CASE THIS^.stSeqCtrlGeneral.eActiveSeqState OF
E_SEQ_GENERAL.READY:;

	
E_SEQ_GENERAL.EXECUTE:;
	IF TRUE
	THEN
		THIS^.stSeqCtrlGeneral.eActiveSeqState := E_SEQ_GENERAL.RESET;
	END_IF
  
E_SEQ_GENERAL.RESET:;
	stSeqCtrlGeneral.iInternalSeqStateCase := 0;
	IF TRUE
	THEN
		THIS^.stSeqCtrlGeneral.eActiveSeqState := E_SEQ_GENERAL.BUSY;
	END_IF
  
E_SEQ_GENERAL.BUSY:;
	CASE THIS^.stSeqCtrlGeneral.iInternalSeqStateCase OF
    0:  // Check state
      IF TRUE
      AND THIS^.itfSensorOpened.P_Active 
      AND THIS^.itfSensorClosed.P_Active 
			THEN 
        THIS^.stSeqCtrlGeneral.eActiveSeqState := E_SEQ_GENERAL.ERROR;
      ELSIF TRUE
      AND THIS^.itfSensorClosed.P_Active
      THEN
        THIS^.stSeqCtrlGeneral.iInternalSeqStateCase := 1000;
      ELSE
        THIS^.itfClose.M_Set();
        THIS^.itfOpen.M_Reset();
        THIS^.stSeqCtrlGeneral.iInternalSeqStateCase := 10;
			END_IF
      
    10: // wait for the end position sensor
      IF TRUE 
			THEN 
        IF TRUE
        AND THIS^.itfSensorClosed.P_Active
        THEN
          THIS^.itfClose.M_Reset();
          THIS^.stSeqCtrlGeneral.iInternalSeqStateCase := 1000;
				END_IF
			END_IF
      
	ELSE
		THIS^.stSeqCtrlGeneral.eActiveSeqState := E_SEQ_GENERAL.DONE;  
	END_CASE
	THIS^.stSeqCtrlGeneral.strExtraInfo := CONCAT('Internal state: ', TO_STRING(THIS^.stSeqCtrlGeneral.iInternalSeqStateCase));

E_SEQ_GENERAL.DONE:;

E_SEQ_GENERAL.ERROR:;

E_SEQ_GENERAL.TIME_OUT:; 
IF TRUE
AND THIS^.stSeqCtrlGeneral.bTimeOutActiveQuit 
THEN
  THIS^.stSeqCtrlGeneral.strExtraInfo := 'Bitte quittieren und erneut testen';
  IF TRUE
  //AND itfOpMode.P_QUIT
  THEN
    THIS^.stSeqCtrlGeneral.eActiveSeqState := E_SEQ_GENERAL.EXECUTE;
	END_IF
  
END_IF

ELSE
  THIS^.stSeqCtrlGeneral.eActiveSeqState := E_SEQ_GENERAL.ERROR;
END_CASE
END_METHOD

METHOD PRIVATE _m_Seq_INIT : BOOL
VAR
  ActiveSeq: STRING;
END_VAR
//THIS^._m_GeneralStepSetting(StepType:=E_STEP_STATE_TYPE.INIT,
ActiveSeq := TO_STRING(THIS^.eSeq);

CASE THIS^.stSeqCtrlGeneral.eActiveSeqState OF
E_SEQ_GENERAL.READY:;

	
E_SEQ_GENERAL.EXECUTE:;
	IF TRUE
	THEN
		THIS^.stSeqCtrlGeneral.eActiveSeqState := E_SEQ_GENERAL.RESET;
	END_IF
  
E_SEQ_GENERAL.RESET:;
	stSeqCtrlGeneral.iInternalSeqStateCase := 0;
	IF TRUE
	THEN
		THIS^.stSeqCtrlGeneral.eActiveSeqState := E_SEQ_GENERAL.BUSY;
	END_IF
  
E_SEQ_GENERAL.BUSY:;
	CASE THIS^.stSeqCtrlGeneral.iInternalSeqStateCase OF
    0:  // Reset valve
      IF TRUE 
			THEN 
        IF THIS^.bNC THEN
          THIS^.itfClose.M_Set();
          THIS^.itfOpen.M_Reset();
        ELSE
          THIS^.itfClose.M_Reset();
          THIS^.itfOpen.M_Set();
				END_IF
        THIS^.stSeqCtrlGeneral.iInternalSeqStateCase := 10;
			END_IF
      
    10: // Wait for the end position sensor
      IF TRUE 
			THEN 
        IF THIS^.bNC 
        AND THIS^.itfSensorClosed.P_Active 
        THEN
          THIS^.itfClose.M_Reset();
          THIS^.stSeqCtrlGeneral.iInternalSeqStateCase := 1000;
        ELSIF NOT THIS^.bNC
        AND THIS^.itfSensorOpened.P_Active
        THEN
          THIS^.itfOpen.M_Reset();
          THIS^.stSeqCtrlGeneral.iInternalSeqStateCase := 1000;
				END_IF
			END_IF
      
	ELSE
		THIS^.stSeqCtrlGeneral.eActiveSeqState := E_SEQ_GENERAL.DONE;  
	END_CASE
	THIS^.stSeqCtrlGeneral.strExtraInfo := CONCAT('Internal state: ', TO_STRING(THIS^.stSeqCtrlGeneral.iInternalSeqStateCase));

E_SEQ_GENERAL.DONE:;

E_SEQ_GENERAL.ERROR:;

E_SEQ_GENERAL.TIME_OUT:; 
IF TRUE
AND THIS^.stSeqCtrlGeneral.bTimeOutActiveQuit 
THEN
  THIS^.stSeqCtrlGeneral.strExtraInfo := 'Bitte quittieren und erneut testen';
  IF TRUE
  //AND itfOpMode.P_QUIT
  THEN
    THIS^.stSeqCtrlGeneral.eActiveSeqState := E_SEQ_GENERAL.EXECUTE;
	END_IF
  
END_IF

ELSE
  THIS^.stSeqCtrlGeneral.eActiveSeqState := E_SEQ_GENERAL.ERROR;
END_CASE
END_METHOD

METHOD PRIVATE _m_Seq_OPEN : BOOL
VAR
  ActiveSeq: STRING;
END_VAR
//THIS^._m_GeneralStepSetting(StepType:=E_STEP_STATE_TYPE.INIT,
ActiveSeq := TO_STRING(THIS^.eSeq);

CASE THIS^.stSeqCtrlGeneral.eActiveSeqState OF
E_SEQ_GENERAL.READY:;

	
E_SEQ_GENERAL.EXECUTE:;
	IF TRUE
	THEN
		THIS^.stSeqCtrlGeneral.eActiveSeqState := E_SEQ_GENERAL.RESET;
	END_IF
  
E_SEQ_GENERAL.RESET:;
	stSeqCtrlGeneral.iInternalSeqStateCase := 0;
	IF TRUE
	THEN
		THIS^.stSeqCtrlGeneral.eActiveSeqState := E_SEQ_GENERAL.BUSY;
	END_IF
  
E_SEQ_GENERAL.BUSY:;
	CASE THIS^.stSeqCtrlGeneral.iInternalSeqStateCase OF
    0:  // Check state
      IF TRUE
      AND THIS^.itfSensorOpened.P_Active 
      AND THIS^.itfSensorClosed.P_Active 
			THEN 
        THIS^.stSeqCtrlGeneral.eActiveSeqState := E_SEQ_GENERAL.ERROR;
      ELSIF TRUE
      AND THIS^.itfSensorOpened.P_Active
      THEN
        THIS^.stSeqCtrlGeneral.iInternalSeqStateCase := 1000;
      ELSE
        THIS^.itfClose.M_Reset();
        THIS^.itfOpen.M_Set();
        THIS^.stSeqCtrlGeneral.iInternalSeqStateCase := 10;
			END_IF
      
    10: // wait for the end position sensor
      IF TRUE 
			THEN 
        IF TRUE
        AND THIS^.itfSensorOpened.P_Active
        THEN
          THIS^.itfOpen.M_Reset();
          THIS^.stSeqCtrlGeneral.iInternalSeqStateCase := 1000;
				END_IF
			END_IF
      
	ELSE
		THIS^.stSeqCtrlGeneral.eActiveSeqState := E_SEQ_GENERAL.DONE;  
	END_CASE
	THIS^.stSeqCtrlGeneral.strExtraInfo := CONCAT('Internal state: ', TO_STRING(THIS^.stSeqCtrlGeneral.iInternalSeqStateCase));

E_SEQ_GENERAL.DONE:;

E_SEQ_GENERAL.ERROR:;

E_SEQ_GENERAL.TIME_OUT:; 
IF TRUE
AND THIS^.stSeqCtrlGeneral.bTimeOutActiveQuit 
THEN
  THIS^.stSeqCtrlGeneral.strExtraInfo := 'Bitte quittieren und erneut testen';
  IF TRUE
  //AND itfOpMode.P_QUIT
  THEN
    THIS^.stSeqCtrlGeneral.eActiveSeqState := E_SEQ_GENERAL.EXECUTE;
	END_IF
  
END_IF

ELSE
  THIS^.stSeqCtrlGeneral.eActiveSeqState := E_SEQ_GENERAL.ERROR;
END_CASE
END_METHOD

METHOD PRIVATE _m_SequenceManager
VAR_INPUT
END_VAR
IF FALSE
//AND THIS^.eActiveSeqState=DONE 
AND eLastSeq<>eSeq
THEN
	IF THIS^.stSeqCtrlGeneral.eActiveSeqState<>E_SEQ_GENERAL.EXECUTE THEN
		THIS^.stSeqCtrlGeneral.eActiveSeqState:=E_SEQ_GENERAL.READY;
	END_IF
END_IF

eSeq := eNextSeq;

//DelayTimer und TimeOut Timer verwalten
stSeqCtrlGeneral.bActiveStep:=	TRUE
				AND eLastSeq					=	eSeq
				AND stSeqCtrlGeneral.eLastActiveSeqState			=	stSeqCtrlGeneral.eActiveSeqState
				AND	stSeqCtrlGeneral.iLastInternalSeqStateCase	=	stSeqCtrlGeneral.iInternalSeqStateCase
				;
			
IF NOT stSeqCtrlGeneral.bActiveStep THEN
	stSeqCtrlGeneral.bDelayActive:=FALSE;
	stSeqCtrlGeneral.bTimeOutActiveQuit:=FALSE;
	stSeqCtrlGeneral.bTimeOutActiveNoQuit:=FALSE;
  THIS^.stSeqCtrlGeneral.strExtraInfo:='';
END_IF

_m_SaveLastStep();
stSeqCtrlGeneral.tonDelay	(IN:=stSeqCtrlGeneral.bActiveStep AND stSeqCtrlGeneral.bDelayActive, 		PT:=stSeqCtrlGeneral.tDelay);
stSeqCtrlGeneral.tonTimeOut	(IN:=stSeqCtrlGeneral.bActiveStep AND (stSeqCtrlGeneral.bTimeOutActiveNoQuit OR stSeqCtrlGeneral.bTimeOutActiveQuit), 	PT:=stSeqCtrlGeneral.tTimeOut);
stSeqCtrlGeneral.tonStepTime	(IN:= stSeqCtrlGeneral.bActiveStep, PT:= T#24H);

IF stSeqCtrlGeneral.tonTimeOut.Q  THEN
	stSeqCtrlGeneral.eActiveSeqState:=E_SEQ_GENERAL.TIME_OUT;
END_IF

IF stSeqCtrlGeneral.iError<>0 THEN
	eSeq:=E_SEQ_ENGINE.ERROR_SEQ;
END_IF



eLastSeq					:=	eSeq;
stSeqCtrlGeneral.eLastActiveSeqState			:=	stSeqCtrlGeneral.eActiveSeqState;
stSeqCtrlGeneral.iLastInternalSeqStateCase	:=	stSeqCtrlGeneral.iInternalSeqStateCase;

// Reset set ready state
IF THIS^.stSeqCtrlGeneral.bExitSetReadyState THEN
  THIS^.stSeqCtrlGeneral.bExitSetReadyState := FALSE;
END_IF
END_METHOD

METHOD PRIVATE _m_TimeOut : BOOL
VAR_INPUT
	bTimeoutActiveToQuit:	BOOL;
	bTimeOutActiveNoQuit:	BOOL;
	tTimeOut:				TIME;	
END_VAR
THIS^.stSeqCtrlGeneral.bTimeOutActiveQuit:=	bTimeoutActiveToQuit;
THIS^.stSeqCtrlGeneral.bTimeOutActiveNoQuit:=	bTimeOutActiveNoQuit;
THIS^.stSeqCtrlGeneral.tTimeOut:=			tTimeOut;
_m_TimeOut:=FALSE;
IF THIS^.stSeqCtrlGeneral.tonTimeOut.Q THEN
	_m_TimeOut:=TRUE;
END_IF
END_METHOD

METHOD FB_init : BOOL
VAR_INPUT
	bInitRetains : BOOL; // if TRUE, the retain variables are initialized (warm start / cold start)
	bInCopyCode : BOOL;  // if TRUE, the instance afterwards gets moved into the copy code (online change)
  
  itfOpMode:											                        I_OP_MODE; 
  itfEventLogger:                                         I_EVENT_LOGGER;
  itfOpen:                                                I_BINARY_OUTPUT;
  itfClose:                                               I_BINARY_OUTPUT;
  itfSensorOpened:                                        I_BINARY_SWITCH;
  itfSensorClosed:                                        I_BINARY_SWITCH;
  bNC:                                                    BOOL;
END_VAR
THIS^.itfOpMode := itfOpMode;
THIS^.itfEventLogger := itfEventLogger;
THIS^.itfOpen := itfOpen;
THIS^.itfClose := itfClose;
THIS^.itfSensorOpened := itfSensorOpened;
THIS^.itfSensorClosed := itfSensorClosed;
THIS^.bNC := bNC;
END_METHOD

METHOD M_Close : BOOL
M_Close := THIS^.stSeqCtrlGeneral.eActiveSeqState = E_SEQ_GENERAL.DONE;

// Assign input

// General
IF THIS^.stSeqCtrlGeneral.eActiveSeqState = E_SEQ_GENERAL.READY THEN
  THIS^.eNextSeq := E_SEQ_ENGINE.CLOSE;
  THIS^.stSeqCtrlGeneral.eActiveSeqState := E_SEQ_GENERAL.EXECUTE;
END_IF
END_METHOD

METHOD M_Open : BOOL
M_Open := THIS^.stSeqCtrlGeneral.eActiveSeqState = E_SEQ_GENERAL.DONE;

// Assign input

// General
IF THIS^.stSeqCtrlGeneral.eActiveSeqState = E_SEQ_GENERAL.READY THEN
  THIS^.eNextSeq := E_SEQ_ENGINE.OPEN;
  THIS^.stSeqCtrlGeneral.eActiveSeqState := E_SEQ_GENERAL.EXECUTE;
END_IF
END_METHOD

METHOD M_Reset : BOOL
VAR_INPUT
END_VAR
M_Reset := THIS^.stSeqCtrlGeneral.eActiveSeqState = E_SEQ_GENERAL.DONE;

// Assign input

// General
IF THIS^.stSeqCtrlGeneral.eActiveSeqState = E_SEQ_GENERAL.READY THEN
  THIS^.eNextSeq := E_SEQ_ENGINE.INIT;
  THIS^.stSeqCtrlGeneral.eActiveSeqState := E_SEQ_GENERAL.EXECUTE;
END_IF
END_METHOD

{warning 'Methodenimplementierung hinzufügen'}
(*=== Method: M_Run  ============================================

 @brief: Here is the global code (Timer, Event, Flange,...)*)
METHOD M_Run
END_METHOD

METHOD M_SetReady : BOOL
VAR_INPUT
END_VAR
M_SetReady := TRUE
              AND THIS^.stSeqCtrlGeneral.eActiveSeqState = E_SEQ_GENERAL.READY
              AND THIS^.eSeq = E_SEQ_VALVE.BASE;

THIS^.stSeqCtrlGeneral.eActiveSeqState := E_SEQ_GENERAL.READY;
THIS^.eNextSeq := E_SEQ_VALVE.BASE;
END_METHOD

PROPERTY P_Closed : BOOL
GET
P_Closed := THIS^.itfSensorClosed.P_Active AND NOT THIS^.itfSensorOpened.P_Active;
END_GET
END_PROPERTY

{warning 'Eigenschaftenimplementierung hinzufügen'}
(*=== Property: P_Event  ============================================

 @param [set]: 	Set the Structure "ST_EVENT" from another Object
 @param [get]: 	Return the Structure "ST_EVENT", it contains the actual 
					event of the Object *)
PROPERTY P_Event : GenLib.ST_EVENT
GET
END_GET
SET
END_SET
END_PROPERTY

{warning 'Eigenschaftenimplementierung hinzufügen'}
(*=== Property: P_FullObjectPath  ============================================

 @param [set]: 	Set the Object Path (Clear String of Object)
 @param [get]: 	Return the Objectpath *)
PROPERTY P_FullObjectPath : STRING
GET
END_GET
SET
END_SET
END_PROPERTY

{warning 'Eigenschaftenimplementierung hinzufügen'}
(*=== Property: P_Global_Ack  ============================================

 @param [set]: 	Set the Bit for Ack from another Object
 @param [get]: 	Return the state of Ack Bit*)
PROPERTY P_Global_Ack : BOOL
GET
END_GET
SET
END_SET
END_PROPERTY

{warning 'Eigenschaftenimplementierung hinzufügen'}
(*=== Property: P_GlobalID  ============================================

 @param [set]: 	-
 @param [get]: 	Return the string of instance path*)
PROPERTY P_GlobalID : STRING
GET
END_GET
END_PROPERTY

{warning 'Eigenschaftenimplementierung hinzufügen'}
PROPERTY P_Open : BOOL
GET
P_Open := NOT THIS^.itfSensorClosed.P_Active AND THIS^.itfSensorOpened.P_Active;
END_GET
END_PROPERTY

{warning 'Eigenschaftenimplementierung hinzufügen'}
PROPERTY P_ReadyState : BOOL
GET
P_ReadyState := THIS^.stSeqCtrlGeneral.eActiveSeqState = E_SEQ_GENERAL.READY;
END_GET
END_PROPERTY

PROPERTY P_Undefined : BOOL
GET
P_Undefined := (NOT THIS^.itfSensorClosed.P_Active AND NOT THIS^.itfSensorOpened.P_Active) OR (THIS^.itfSensorClosed.P_Active AND THIS^.itfSensorOpened.P_Active);
END_GET
END_PROPERTY

END_FUNCTION_BLOCK

// ---- MODULE/ACTOR_VALVE/VALVE/POU/FB_VALVE_X_2.TcPOU
FUNCTION_BLOCK FB_VALVE_X_2 IMPLEMENTS I_VALVE_X_2
VAR //General
	{attribute 'instance-path'} 
  {attribute 'noinit'} 
	strInstancePath:									                      STRING;
	bInit: 												                          BOOL:=TRUE;
	strFullObjectPath: 								                      STRING;
	stEvent:											                          ST_EVENT;
	bAck:												                            BOOL;
	
END_VAR
VAR   // From FB_init	
	itfOpMode:											                        I_OP_MODE; 
  itfEventLogger:                                         I_EVENT_LOGGER;
  itfSwitchToWP:                                          I_BINARY_OUTPUT;
END_VAR                                      				
VAR	// Step chain control                				
  eSeq, eLastSeq, eNextSeq:					                      E_SEQ_VALVE; 
                  				
  //eActiveSeqState, eLastActiveSeqState:                 E_SEQ_GENERAL;
	(*
  iInternalSeqStateCase, iLastInternalSeqStateCase:       INT:=0;       
	tonDelay, tonTimeOut, tonStepTime:						          TON;
	tDelay:													                        TIME := T#100MS;
	tTimeOut:												                        TIME := T#100MS;
	tTimeOutExt:											                      TIME := T#100MS;
	bDelayActive, bTimeOutActiveQuit, bTimeOutActiveNoQuit:	BOOL;//Timer Option
	bActiveStep, bDebugAcitve, bDebugNext:					        BOOL;//Debug Option
	i:														                          INT;
 	iError:													                        INT; //ERROR-CODE                    	                   		
	listLastSteps:											                    ARRAY[0..49] OF ST_LAST_STEPS;	
	strExtraInfo:											                      STRING; 
	eStep_Type:												                      E_STEP_STATE_TYPE; 
	bDebugModeActive:										                    BOOL;   
	bWaitForBreakpoint:										                  BOOL;
	bBreakpointActive:										                  BOOL;
	bDebugResume:											                      BOOL;   
	listBreakpoint:											                    ARRAY[0..10] OF  INT;    
*)
i:														                            INT;
stSeqCtrlGeneral:											                    ST_SEQ_CTRL_GEN;     	
END_VAR                                             		
VAR                                                 		
	bMethodeFromExtStarted:									                BOOL;
	bMethodeFromExtActive:									                BOOL;
	bMethodeFromExtDone:									                  BOOL;
	strTemp:												                        STRING;
END_VAR   
VAR
  stHMI:                                                  ST_HMI_VALVE;
  tDelay:                                                 TIME;
END_VAR                  	
VAR_TEMP                    	
	iTemp:										                              INT;
END_VAR

// Set FBs and Interfaces ready after switch internal step
IF stSeqCtrlGeneral.iInternalSeqStateCase <> stSeqCtrlGeneral.iLastInternalSeqStateCase AND NOT stSeqCtrlGeneral.bExitSetReadyState THEN
  IF TRUE
  //AND ...
  THEN
    stSeqCtrlGeneral.bExitSetReadyState := TRUE;
  ELSE
    RETURN;
  END_IF
END_IF

stSeqCtrlGeneral.strObject := F_CreateObjectName(strInstancePath);

// First method call
_m_SequenceManager();
//_m_SaveLastStep();

CASE eSeq OF 
  E_SEQ_VALVE.BASE:;
  
	E_SEQ_VALVE.INIT: _m_Seq_INIT();
		IF TRUE
		AND (stSeqCtrlGeneral.eActiveSeqState = E_SEQ_GENERAL.DONE) 
		THEN
			eSeq := E_SEQ_VALVE.BASE;
		END_IF
		
	E_SEQ_VALVE.SETUP:;
  
	// Process
  E_SEQ_VALVE.SET_HP: _m_Seq_TO_HP();
    IF TRUE
		AND (stSeqCtrlGeneral.eActiveSeqState = E_SEQ_GENERAL.DONE) 
		THEN
			eSeq := E_SEQ_VALVE.BASE;
		END_IF
  
	E_SEQ_VALVE.SET_WP1:  _m_Seq_TO_WP1();
    IF TRUE
		AND (stSeqCtrlGeneral.eActiveSeqState = E_SEQ_GENERAL.DONE) 
		THEN
			eSeq := E_SEQ_VALVE.BASE;
		END_IF

  // End
	E_SEQ_VALVE.END:;
	E_SEQ_VALVE.ERROR_SEQ:;	
END_CASE

strTemp:=TO_STRING(eSeq);

METHOD PRIVATE _m_DebugManager
VAR_INPUT
	iStepID: int;
END_VAR
IF TRUE
AND THIS^.stSeqCtrlGeneral.bDebugModeActive 
AND NOT THIS^.stSeqCtrlGeneral.bActiveStep
THEN


THIS^.stSeqCtrlGeneral.bBreakpointActive:=FALSE;

FOR i:=0 TO 10 DO
	
	IF TRUE
	AND iStepID=THIS^.stSeqCtrlGeneral.listBreakpoint[i] 
	AND iStepID<>0
	THEN
		EXIT;
	END_IF
END_FOR
IF (i<=10) THEN
	THIS^.stSeqCtrlGeneral.bBreakpointActive:=TRUE;
END_IF

END_IF
END_METHOD

METHOD PRIVATE _m_Delay : BOOL
VAR_INPUT
	DelayTime:	TIME;
END_VAR
THIS^.stSeqCtrlGeneral.bDelayActive:=TRUE;
THIS^.stSeqCtrlGeneral.tDelay:=DelayTime;
_m_Delay:=FALSE;
IF THIS^.stSeqCtrlGeneral.tonDelay.Q THEN
	_m_Delay:=TRUE;
END_IF
END_METHOD

METHOD PRIVATE _m_GeneralStepSetting : BOOL
VAR_INPUT
	StepType:			    	E_STEP_STATE_TYPE;
	InfoTextID:					STRING(20);
	EnableDebug:	   			BOOL;	
	
END_VAR
IF THIS^.stSeqCtrlGeneral.bActiveStep THEN
	THIS^.stSeqCtrlGeneral.eStep_Type:=StepType;
	THIS^.stSeqCtrlGeneral.strExtraInfo:= GenLib.F_RET_TXTLIST_ENTRY(strPortNr:='851',strID:='',strTxtLstName:=InfoTextID);
END_IF
END_METHOD

METHOD PRIVATE _m_SaveLastStep : BOOL
VAR_INPUT
END_VAR
VAR
	i: dint;
END_VAR
IF NOT THIS^.stSeqCtrlGeneral.bActiveStep THEN
	
	FOR i:=49 TO 1 BY -1 DO
			stSeqCtrlGeneral.listLastSteps[i].strStepName:=stSeqCtrlGeneral.listLastSteps[i-1].strStepName;
			stSeqCtrlGeneral.listLastSteps[i].tStepTime:=stSeqCtrlGeneral.listLastSteps[i-1].tStepTime;
			stSeqCtrlGeneral.listLastSteps[i].tDelayTime:=stSeqCtrlGeneral.listLastSteps[i-1].tDelayTime;
	END_FOR
	stSeqCtrlGeneral.listLastSteps[0].strStepName:=TO_STRING(THIS^.eSeq);
	stSeqCtrlGeneral.listLastSteps[1].tStepTime:=THIS^.stSeqCtrlGeneral.tonStepTime.ET;
	stSeqCtrlGeneral.listLastSteps[1].tStepTime:=THIS^.stSeqCtrlGeneral.tonDelay.ET;
ELSE
	stSeqCtrlGeneral.listLastSteps[0].tStepTime:=THIS^.stSeqCtrlGeneral.tonStepTime.ET;
	stSeqCtrlGeneral.listLastSteps[0].tDelayTime:=THIS^.stSeqCtrlGeneral.tonDelay.ET;	
END_IF
END_METHOD

METHOD PRIVATE _m_Seq_INIT : BOOL
VAR
  ActiveSeq: STRING;
END_VAR
//THIS^._m_GeneralStepSetting(StepType:=E_STEP_STATE_TYPE.INIT,
ActiveSeq := TO_STRING(THIS^.eSeq);

CASE THIS^.stSeqCtrlGeneral.eActiveSeqState OF
E_SEQ_GENERAL.READY:;

	
E_SEQ_GENERAL.EXECUTE:;
	IF TRUE
	THEN
		THIS^.stSeqCtrlGeneral.eActiveSeqState := E_SEQ_GENERAL.RESET;
	END_IF
  
E_SEQ_GENERAL.RESET:;
	stSeqCtrlGeneral.iInternalSeqStateCase := 0;
	IF TRUE
	THEN
		THIS^.stSeqCtrlGeneral.eActiveSeqState := E_SEQ_GENERAL.BUSY;
	END_IF
  
E_SEQ_GENERAL.BUSY:;
	CASE THIS^.stSeqCtrlGeneral.iInternalSeqStateCase OF
    0:  // Reset valve
      IF TRUE 
			THEN 
        itfSwitchToWP.M_Reset();
        IF _m_Delay(T#1S) THEN
          THIS^.stSeqCtrlGeneral.iInternalSeqStateCase := 1000;
				END_IF
      ELSE
        THIS^.stSeqCtrlGeneral.eActiveSeqState := E_SEQ_GENERAL.ERROR;
			END_IF
      
	ELSE
		THIS^.stSeqCtrlGeneral.eActiveSeqState := E_SEQ_GENERAL.DONE;  
	END_CASE
	THIS^.stSeqCtrlGeneral.strExtraInfo := CONCAT('Internal state: ', TO_STRING(THIS^.stSeqCtrlGeneral.iInternalSeqStateCase));

E_SEQ_GENERAL.DONE:;

E_SEQ_GENERAL.ERROR:;

E_SEQ_GENERAL.TIME_OUT:; 
IF TRUE
AND THIS^.stSeqCtrlGeneral.bTimeOutActiveQuit 
THEN
  THIS^.stSeqCtrlGeneral.strExtraInfo := 'Bitte quittieren und erneut testen';
  IF TRUE
  //AND itfOpMode.P_QUIT
  THEN
    THIS^.stSeqCtrlGeneral.eActiveSeqState := E_SEQ_GENERAL.EXECUTE;
	END_IF
  
END_IF

ELSE
  THIS^.stSeqCtrlGeneral.eActiveSeqState := E_SEQ_GENERAL.ERROR;
END_CASE
END_METHOD

METHOD PRIVATE _m_Seq_TO_HP : BOOL
VAR
  ActiveSeq: STRING;
END_VAR
//THIS^._m_GeneralStepSetting(StepType:=E_STEP_STATE_TYPE.INIT,
ActiveSeq := TO_STRING(THIS^.eSeq);

CASE THIS^.stSeqCtrlGeneral.eActiveSeqState OF
E_SEQ_GENERAL.READY:;

	
E_SEQ_GENERAL.EXECUTE:;
	IF TRUE
	THEN
		THIS^.stSeqCtrlGeneral.eActiveSeqState := E_SEQ_GENERAL.RESET;
	END_IF
  
E_SEQ_GENERAL.RESET:;
	stSeqCtrlGeneral.iInternalSeqStateCase := 0;
	IF TRUE
	THEN
		THIS^.stSeqCtrlGeneral.eActiveSeqState := E_SEQ_GENERAL.BUSY;
	END_IF
  
E_SEQ_GENERAL.BUSY:;
	CASE THIS^.stSeqCtrlGeneral.iInternalSeqStateCase OF
    0:  // Reset valve
      IF TRUE 
			THEN 
        itfSwitchToWP.M_Reset();
        IF _m_Delay(tDelay) THEN
          THIS^.stSeqCtrlGeneral.iInternalSeqStateCase := 1000;
				END_IF
			END_IF
      
	ELSE
		THIS^.stSeqCtrlGeneral.eActiveSeqState := E_SEQ_GENERAL.DONE;  
	END_CASE
	THIS^.stSeqCtrlGeneral.strExtraInfo := CONCAT('Internal state: ', TO_STRING(THIS^.stSeqCtrlGeneral.iInternalSeqStateCase));

E_SEQ_GENERAL.DONE:;

E_SEQ_GENERAL.ERROR:;

E_SEQ_GENERAL.TIME_OUT:; 
IF TRUE
AND THIS^.stSeqCtrlGeneral.bTimeOutActiveQuit 
THEN
  THIS^.stSeqCtrlGeneral.strExtraInfo := 'Bitte quittieren und erneut testen';
  IF TRUE
  //AND itfOpMode.P_QUIT
  THEN
    THIS^.stSeqCtrlGeneral.eActiveSeqState := E_SEQ_GENERAL.EXECUTE;
	END_IF
  
END_IF

ELSE
  THIS^.stSeqCtrlGeneral.eActiveSeqState := E_SEQ_GENERAL.ERROR;
END_CASE
END_METHOD

METHOD PRIVATE _m_Seq_TO_WP1 : BOOL
VAR
  ActiveSeq: STRING;
END_VAR
//THIS^._m_GeneralStepSetting(StepType:=E_STEP_STATE_TYPE.INIT,
ActiveSeq := TO_STRING(THIS^.eSeq);

CASE THIS^.stSeqCtrlGeneral.eActiveSeqState OF
E_SEQ_GENERAL.READY:;

	
E_SEQ_GENERAL.EXECUTE:;
	IF TRUE
	THEN
		THIS^.stSeqCtrlGeneral.eActiveSeqState := E_SEQ_GENERAL.RESET;
	END_IF
  
E_SEQ_GENERAL.RESET:;
	stSeqCtrlGeneral.iInternalSeqStateCase := 0;
	IF TRUE
	THEN
		THIS^.stSeqCtrlGeneral.eActiveSeqState := E_SEQ_GENERAL.BUSY;
	END_IF
  
E_SEQ_GENERAL.BUSY:;
	CASE THIS^.stSeqCtrlGeneral.iInternalSeqStateCase OF
    0:  // Reset valve
      IF TRUE 
			THEN 
        itfSwitchToWP.M_Set();
        IF _m_Delay(tDelay) THEN
          THIS^.stSeqCtrlGeneral.iInternalSeqStateCase := 1000;
				END_IF
			END_IF
      
	ELSE
		THIS^.stSeqCtrlGeneral.eActiveSeqState := E_SEQ_GENERAL.DONE;  
	END_CASE
	THIS^.stSeqCtrlGeneral.strExtraInfo := CONCAT('Internal state: ', TO_STRING(THIS^.stSeqCtrlGeneral.iInternalSeqStateCase));

E_SEQ_GENERAL.DONE:;

E_SEQ_GENERAL.ERROR:;

E_SEQ_GENERAL.TIME_OUT:; 
IF TRUE
AND THIS^.stSeqCtrlGeneral.bTimeOutActiveQuit 
THEN
  THIS^.stSeqCtrlGeneral.strExtraInfo := 'Bitte quittieren und erneut testen';
  IF TRUE
  //AND itfOpMode.P_QUIT
  THEN
    THIS^.stSeqCtrlGeneral.eActiveSeqState := E_SEQ_GENERAL.EXECUTE;
	END_IF
  
END_IF

ELSE
  THIS^.stSeqCtrlGeneral.eActiveSeqState := E_SEQ_GENERAL.ERROR;
END_CASE
END_METHOD

METHOD PRIVATE _m_SequenceManager
VAR_INPUT
END_VAR
IF FALSE
//AND THIS^.eActiveSeqState=DONE 
AND eLastSeq<>eSeq
THEN
	IF THIS^.stSeqCtrlGeneral.eActiveSeqState<>E_SEQ_GENERAL.EXECUTE THEN
		THIS^.stSeqCtrlGeneral.eActiveSeqState:=E_SEQ_GENERAL.READY;
	END_IF
END_IF

eSeq := eNextSeq;

//DelayTimer und TimeOut Timer verwalten
stSeqCtrlGeneral.bActiveStep:=	TRUE
				AND eLastSeq					=	eSeq
				AND stSeqCtrlGeneral.eLastActiveSeqState			=	stSeqCtrlGeneral.eActiveSeqState
				AND	stSeqCtrlGeneral.iLastInternalSeqStateCase	=	stSeqCtrlGeneral.iInternalSeqStateCase
				;
			
IF NOT stSeqCtrlGeneral.bActiveStep THEN
	stSeqCtrlGeneral.bDelayActive:=FALSE;
	stSeqCtrlGeneral.bTimeOutActiveQuit:=FALSE;
	stSeqCtrlGeneral.bTimeOutActiveNoQuit:=FALSE;
  THIS^.stSeqCtrlGeneral.strExtraInfo:='';
END_IF

_m_SaveLastStep();
stSeqCtrlGeneral.tonDelay	(IN:=stSeqCtrlGeneral.bActiveStep AND stSeqCtrlGeneral.bDelayActive, 		PT:=stSeqCtrlGeneral.tDelay);
stSeqCtrlGeneral.tonTimeOut	(IN:=stSeqCtrlGeneral.bActiveStep AND (stSeqCtrlGeneral.bTimeOutActiveNoQuit OR stSeqCtrlGeneral.bTimeOutActiveQuit), 	PT:=stSeqCtrlGeneral.tTimeOut);
stSeqCtrlGeneral.tonStepTime	(IN:= stSeqCtrlGeneral.bActiveStep, PT:= T#24H);

IF stSeqCtrlGeneral.tonTimeOut.Q  THEN
	stSeqCtrlGeneral.eActiveSeqState:=E_SEQ_GENERAL.TIME_OUT;
END_IF

IF stSeqCtrlGeneral.iError<>0 THEN
	eSeq:=E_SEQ_VALVE.ERROR_SEQ;
END_IF



eLastSeq					:=	eSeq;
stSeqCtrlGeneral.eLastActiveSeqState			:=	stSeqCtrlGeneral.eActiveSeqState;
stSeqCtrlGeneral.iLastInternalSeqStateCase	:=	stSeqCtrlGeneral.iInternalSeqStateCase;

// Reset set ready state
IF THIS^.stSeqCtrlGeneral.bExitSetReadyState THEN
  THIS^.stSeqCtrlGeneral.bExitSetReadyState := FALSE;
END_IF
END_METHOD

METHOD PRIVATE _m_TimeOut : BOOL
VAR_INPUT
	bTimeoutActiveToQuit:	BOOL;
	bTimeOutActiveNoQuit:	BOOL;
	tTimeOut:				TIME;	
END_VAR
THIS^.stSeqCtrlGeneral.bTimeOutActiveQuit:=	bTimeoutActiveToQuit;
THIS^.stSeqCtrlGeneral.bTimeOutActiveNoQuit:=	bTimeOutActiveNoQuit;
THIS^.stSeqCtrlGeneral.tTimeOut:=			tTimeOut;
_m_TimeOut:=FALSE;
IF THIS^.stSeqCtrlGeneral.tonTimeOut.Q THEN
	_m_TimeOut:=TRUE;
END_IF
END_METHOD

METHOD FB_init : BOOL
VAR_INPUT
	bInitRetains : BOOL; // if TRUE, the retain variables are initialized (warm start / cold start)
	bInCopyCode : BOOL;  // if TRUE, the instance afterwards gets moved into the copy code (online change)
  
  itfOpMode:											                        I_OP_MODE;
  itfEventLogger:                                         I_EVENT_LOGGER;
  itfSwitchToWP:                                          I_BINARY_OUTPUT;
END_VAR
THIS^.itfOpMode := itfOpMode;
THIS^.itfEventLogger := itfEventLogger;
THIS^.itfSwitchToWP := itfSwitchToWP;
END_METHOD

METHOD M_Reset : BOOL
VAR_INPUT
END_VAR
M_Reset := THIS^.stSeqCtrlGeneral.eActiveSeqState = E_SEQ_GENERAL.DONE;

// Assign input

// General
IF THIS^.stSeqCtrlGeneral.eActiveSeqState = E_SEQ_GENERAL.READY THEN
  THIS^.eNextSeq := E_SEQ_VALVE.INIT;
  THIS^.stSeqCtrlGeneral.eActiveSeqState := E_SEQ_GENERAL.EXECUTE;
END_IF
END_METHOD

(*=== Method: M_Run  ============================================

 @brief: Here is the global code (Timer, Event, Flange,...)*)
METHOD M_Run
END_METHOD

METHOD M_SetReady : BOOL
VAR_INPUT
END_VAR
M_SetReady := TRUE
              AND THIS^.stSeqCtrlGeneral.eActiveSeqState = E_SEQ_GENERAL.READY
              AND THIS^.eSeq = E_SEQ_VALVE.BASE;

THIS^.stSeqCtrlGeneral.eActiveSeqState := E_SEQ_GENERAL.READY;
THIS^.eNextSeq := E_SEQ_VALVE.BASE;
END_METHOD

METHOD M_ToHP : BOOL
VAR_INPUT
  tDelay:         TIME;
END_VAR
M_ToHP := THIS^.stSeqCtrlGeneral.eActiveSeqState = E_SEQ_GENERAL.DONE;

// Assign input
THIS^.tDelay := tDelay;

// General
IF THIS^.stSeqCtrlGeneral.eActiveSeqState = E_SEQ_GENERAL.READY THEN
  THIS^.eNextSeq := E_SEQ_VALVE.SET_HP;
  THIS^.stSeqCtrlGeneral.eActiveSeqState := E_SEQ_GENERAL.EXECUTE;
END_IF
END_METHOD

METHOD M_ToWP1 : BOOL
VAR_INPUT
  tDelay:        TIME;
END_VAR
M_ToWP1 := THIS^.stSeqCtrlGeneral.eActiveSeqState = E_SEQ_GENERAL.DONE;

// Assign input
THIS^.tDelay := tDelay;

// General
IF THIS^.stSeqCtrlGeneral.eActiveSeqState = E_SEQ_GENERAL.READY THEN
  THIS^.eNextSeq := E_SEQ_VALVE.SET_WP1;
  THIS^.stSeqCtrlGeneral.eActiveSeqState := E_SEQ_GENERAL.EXECUTE;
END_IF
END_METHOD

(*=== Property: P_Event  ============================================

 @param [set]: 	Set the Structure "ST_EVENT" from another Object
 @param [get]: 	Return the Structure "ST_EVENT", it contains the actual 
					event of the Object *)
PROPERTY P_Event : GenLib.ST_EVENT
GET
END_GET
SET
END_SET
END_PROPERTY

{warning 'Eigenschaftenimplementierung hinzufügen'}
(*=== Property: P_FullObjectPath  ============================================

 @param [set]: 	Set the Object Path (Clear String of Object)
 @param [get]: 	Return the Objectpath *)
PROPERTY P_FullObjectPath : STRING
GET
END_GET
SET
END_SET
END_PROPERTY

{warning 'Eigenschaftenimplementierung hinzufügen'}
(*=== Property: P_Global_Ack  ============================================

 @param [set]: 	Set the Bit for Ack from another Object
 @param [get]: 	Return the state of Ack Bit*)
PROPERTY P_Global_Ack : BOOL
GET
END_GET
SET
END_SET
END_PROPERTY

{warning 'Eigenschaftenimplementierung hinzufügen'}
(*=== Property: P_GlobalID  ============================================

 @param [set]: 	-
 @param [get]: 	Return the string of instance path*)
PROPERTY P_GlobalID : STRING
GET
END_GET
END_PROPERTY

PROPERTY P_InHP : BOOL
GET
P_InHP := NOT THIS^.itfSwitchToWP.P_State;
END_GET
END_PROPERTY

PROPERTY P_InWP1 : BOOL
GET
P_InWP1 := THIS^.itfSwitchToWP.P_State;
END_GET
END_PROPERTY

{warning 'Eigenschaftenimplementierung hinzufügen'}
PROPERTY P_ReadyState : BOOL
GET
P_ReadyState := THIS^.stSeqCtrlGeneral.eActiveSeqState = E_SEQ_GENERAL.READY;
END_GET
END_PROPERTY

END_FUNCTION_BLOCK

// ---- MODULE/ACTOR_VALVE/VALVE/POU/FB_VALVE_X_3.TcPOU
FUNCTION_BLOCK FB_VALVE_X_3 IMPLEMENTS I_VALVE_X_3
VAR //General
	{attribute 'instance-path'} 
  {attribute 'noinit'} 
	strInstancePath:									                      STRING;
	bInit: 												                          BOOL:=TRUE;
	strFullObjectPath: 								                      STRING;
	stEvent:											                          ST_EVENT;
	bAck:												                            BOOL;
	
END_VAR
VAR   // From FB_init	
	itfOpMode:											                        I_OP_MODE;
  itfEventLogger:                                         I_EVENT_LOGGER;
  itfSwitchToWP1:                                         I_BINARY_OUTPUT;
  itfSwitchToWP2:                                         I_BINARY_OUTPUT;
END_VAR                                      				
VAR	// Step chain control                				
  eSeq, eLastSeq, eNextSeq:					                      E_SEQ_VALVE; 
                  				
  //eActiveSeqState, eLastActiveSeqState:                 E_SEQ_GENERAL;
	(*
  iInternalSeqStateCase, iLastInternalSeqStateCase:       INT:=0;       
	tonDelay, tonTimeOut, tonStepTime:						          TON;
	tDelay:													                        TIME := T#100MS;
	tTimeOut:												                        TIME := T#100MS;
	tTimeOutExt:											                      TIME := T#100MS;
	bDelayActive, bTimeOutActiveQuit, bTimeOutActiveNoQuit:	BOOL;//Timer Option
	bActiveStep, bDebugAcitve, bDebugNext:					        BOOL;//Debug Option
	i:														                          INT;
 	iError:													                        INT; //ERROR-CODE                    	                   		
	listLastSteps:											                    ARRAY[0..49] OF ST_LAST_STEPS;	
	strExtraInfo:											                      STRING; 
	eStep_Type:												                      E_STEP_STATE_TYPE; 
	bDebugModeActive:										                    BOOL;   
	bWaitForBreakpoint:										                  BOOL;
	bBreakpointActive:										                  BOOL;
	bDebugResume:											                      BOOL;   
	listBreakpoint:											                    ARRAY[0..10] OF  INT;    
*)
i:														                            INT;
stSeqCtrlGeneral:											                    ST_SEQ_CTRL_GEN;     	
END_VAR                                             		
VAR                                                 		
	bMethodeFromExtStarted:									                BOOL;
	bMethodeFromExtActive:									                BOOL;
	bMethodeFromExtDone:									                  BOOL;
	strTemp:												                        STRING;
END_VAR   
VAR
  stHMI:                                                  ST_HMI_VALVE;
  tDelay:                                                 TIME;
END_VAR                  	
VAR_TEMP                    	
	iTemp:										                              INT;
END_VAR

// Set FBs and Interfaces ready after switch internal step
IF stSeqCtrlGeneral.iInternalSeqStateCase <> stSeqCtrlGeneral.iLastInternalSeqStateCase AND NOT stSeqCtrlGeneral.bExitSetReadyState THEN
  IF TRUE
  //AND ...
  THEN
    stSeqCtrlGeneral.bExitSetReadyState := TRUE;
  ELSE
    RETURN;
  END_IF
END_IF

stSeqCtrlGeneral.strObject := F_CreateObjectName(strInstancePath);

// First method call
_m_SequenceManager();
//_m_SaveLastStep();

CASE eSeq OF 
  E_SEQ_VALVE.BASE:;
  
	E_SEQ_VALVE.INIT: _m_Seq_INIT();
		IF TRUE
		AND (stSeqCtrlGeneral.eActiveSeqState = E_SEQ_GENERAL.DONE) 
		THEN
			eSeq := E_SEQ_VALVE.BASE;
		END_IF
		
	E_SEQ_VALVE.SETUP:;
  
	// Process
  E_SEQ_VALVE.SET_HP: _m_Seq_TO_HP();
    IF TRUE
		AND (stSeqCtrlGeneral.eActiveSeqState = E_SEQ_GENERAL.DONE) 
		THEN
			eSeq := E_SEQ_VALVE.BASE;
		END_IF
  
	E_SEQ_VALVE.SET_WP1:  _m_Seq_TO_WP1();
    IF TRUE
		AND (stSeqCtrlGeneral.eActiveSeqState = E_SEQ_GENERAL.DONE) 
		THEN
			eSeq := E_SEQ_VALVE.BASE;
		END_IF
    
  E_SEQ_VALVE.SET_WP2: _m_Seq_TO_WP2();
    IF TRUE
		AND (stSeqCtrlGeneral.eActiveSeqState = E_SEQ_GENERAL.DONE) 
		THEN
			eSeq := E_SEQ_VALVE.BASE;
		END_IF

  // End
	E_SEQ_VALVE.END:;
	E_SEQ_VALVE.ERROR_SEQ:;	
END_CASE

strTemp:=TO_STRING(eSeq);

METHOD PRIVATE _m_DebugManager
VAR_INPUT
	iStepID: int;
END_VAR
IF TRUE
AND THIS^.stSeqCtrlGeneral.bDebugModeActive 
AND NOT THIS^.stSeqCtrlGeneral.bActiveStep
THEN


THIS^.stSeqCtrlGeneral.bBreakpointActive:=FALSE;

FOR i:=0 TO 10 DO
	
	IF TRUE
	AND iStepID=THIS^.stSeqCtrlGeneral.listBreakpoint[i] 
	AND iStepID<>0
	THEN
		EXIT;
	END_IF
END_FOR
IF (i<=10) THEN
	THIS^.stSeqCtrlGeneral.bBreakpointActive:=TRUE;
END_IF

END_IF
END_METHOD

METHOD PRIVATE _m_Delay : BOOL
VAR_INPUT
	DelayTime:	TIME;
END_VAR
THIS^.stSeqCtrlGeneral.bDelayActive:=TRUE;
THIS^.stSeqCtrlGeneral.tDelay:=DelayTime;
_m_Delay:=FALSE;
IF THIS^.stSeqCtrlGeneral.tonDelay.Q THEN
	_m_Delay:=TRUE;
END_IF
END_METHOD

METHOD PRIVATE _m_GeneralStepSetting : BOOL
VAR_INPUT
	StepType:			    	E_STEP_STATE_TYPE;
	InfoTextID:					STRING(20);
	EnableDebug:	   			BOOL;	
	
END_VAR
IF THIS^.stSeqCtrlGeneral.bActiveStep THEN
	THIS^.stSeqCtrlGeneral.eStep_Type:=StepType;
	THIS^.stSeqCtrlGeneral.strExtraInfo:= GenLib.F_RET_TXTLIST_ENTRY(strPortNr:='851',strID:='',strTxtLstName:=InfoTextID);
END_IF
END_METHOD

METHOD PRIVATE _m_SaveLastStep : BOOL
VAR_INPUT
END_VAR
VAR
	i: dint;
END_VAR
IF NOT THIS^.stSeqCtrlGeneral.bActiveStep THEN
	
	FOR i:=49 TO 1 BY -1 DO
			stSeqCtrlGeneral.listLastSteps[i].strStepName:=stSeqCtrlGeneral.listLastSteps[i-1].strStepName;
			stSeqCtrlGeneral.listLastSteps[i].tStepTime:=stSeqCtrlGeneral.listLastSteps[i-1].tStepTime;
			stSeqCtrlGeneral.listLastSteps[i].tDelayTime:=stSeqCtrlGeneral.listLastSteps[i-1].tDelayTime;
	END_FOR
	stSeqCtrlGeneral.listLastSteps[0].strStepName:=TO_STRING(THIS^.eSeq);
	stSeqCtrlGeneral.listLastSteps[1].tStepTime:=THIS^.stSeqCtrlGeneral.tonStepTime.ET;
	stSeqCtrlGeneral.listLastSteps[1].tStepTime:=THIS^.stSeqCtrlGeneral.tonDelay.ET;
ELSE
	stSeqCtrlGeneral.listLastSteps[0].tStepTime:=THIS^.stSeqCtrlGeneral.tonStepTime.ET;
	stSeqCtrlGeneral.listLastSteps[0].tDelayTime:=THIS^.stSeqCtrlGeneral.tonDelay.ET;	
END_IF
END_METHOD

METHOD PRIVATE _m_Seq_INIT : BOOL
VAR
  ActiveSeq: STRING;
END_VAR
//THIS^._m_GeneralStepSetting(StepType:=E_STEP_STATE_TYPE.INIT,
ActiveSeq := TO_STRING(THIS^.eSeq);

CASE THIS^.stSeqCtrlGeneral.eActiveSeqState OF
E_SEQ_GENERAL.READY:;

	
E_SEQ_GENERAL.EXECUTE:;
	IF TRUE
	THEN
		THIS^.stSeqCtrlGeneral.eActiveSeqState := E_SEQ_GENERAL.RESET;
	END_IF
  
E_SEQ_GENERAL.RESET:;
	stSeqCtrlGeneral.iInternalSeqStateCase := 0;
	IF TRUE
	THEN
		THIS^.stSeqCtrlGeneral.eActiveSeqState := E_SEQ_GENERAL.BUSY;
	END_IF
  
E_SEQ_GENERAL.BUSY:;
	CASE THIS^.stSeqCtrlGeneral.iInternalSeqStateCase OF
    0:  // Reset valve
      IF TRUE
			THEN 
        itfSwitchToWP1.M_Reset();
        itfSwitchToWP2.M_Reset();
        IF _m_Delay(T#1S) THEN
          THIS^.stSeqCtrlGeneral.iInternalSeqStateCase := 1000;
				END_IF
			END_IF
      
	ELSE
		THIS^.stSeqCtrlGeneral.eActiveSeqState := E_SEQ_GENERAL.DONE;  
	END_CASE
	THIS^.stSeqCtrlGeneral.strExtraInfo := CONCAT('Internal state: ', TO_STRING(THIS^.stSeqCtrlGeneral.iInternalSeqStateCase));

E_SEQ_GENERAL.DONE:;

E_SEQ_GENERAL.ERROR:;

E_SEQ_GENERAL.TIME_OUT:; 
IF TRUE
AND THIS^.stSeqCtrlGeneral.bTimeOutActiveQuit 
THEN
  THIS^.stSeqCtrlGeneral.strExtraInfo := 'Bitte quittieren und erneut testen';
  IF TRUE
  //AND itfOpMode.P_QUIT
  THEN
    THIS^.stSeqCtrlGeneral.eActiveSeqState := E_SEQ_GENERAL.EXECUTE;
	END_IF
  
END_IF

ELSE
  THIS^.stSeqCtrlGeneral.eActiveSeqState := E_SEQ_GENERAL.ERROR;
END_CASE
END_METHOD

METHOD PRIVATE _m_Seq_TO_HP : BOOL
VAR
  ActiveSeq: STRING;
END_VAR
//THIS^._m_GeneralStepSetting(StepType:=E_STEP_STATE_TYPE.INIT,
ActiveSeq := TO_STRING(THIS^.eSeq);

CASE THIS^.stSeqCtrlGeneral.eActiveSeqState OF
E_SEQ_GENERAL.READY:;

	
E_SEQ_GENERAL.EXECUTE:;
	IF TRUE
	THEN
		THIS^.stSeqCtrlGeneral.eActiveSeqState := E_SEQ_GENERAL.RESET;
	END_IF
  
E_SEQ_GENERAL.RESET:;
	stSeqCtrlGeneral.iInternalSeqStateCase := 0;
	IF TRUE
	THEN
		THIS^.stSeqCtrlGeneral.eActiveSeqState := E_SEQ_GENERAL.BUSY;
	END_IF
  
E_SEQ_GENERAL.BUSY:;
	CASE THIS^.stSeqCtrlGeneral.iInternalSeqStateCase OF
    0:  // Reset valve
      IF TRUE 
			THEN 
        itfSwitchToWP1.M_Reset();
        itfSwitchToWP2.M_Reset();
        IF _m_Delay(tDelay) THEN
          THIS^.stSeqCtrlGeneral.iInternalSeqStateCase := 1000;
				END_IF
			END_IF
      
	ELSE
		THIS^.stSeqCtrlGeneral.eActiveSeqState := E_SEQ_GENERAL.DONE;  
	END_CASE
	THIS^.stSeqCtrlGeneral.strExtraInfo := CONCAT('Internal state: ', TO_STRING(THIS^.stSeqCtrlGeneral.iInternalSeqStateCase));

E_SEQ_GENERAL.DONE:;

E_SEQ_GENERAL.ERROR:;

E_SEQ_GENERAL.TIME_OUT:; 
IF TRUE
AND THIS^.stSeqCtrlGeneral.bTimeOutActiveQuit 
THEN
  THIS^.stSeqCtrlGeneral.strExtraInfo := 'Bitte quittieren und erneut testen';
  IF TRUE
  //AND itfOpMode.P_QUIT
  THEN
    THIS^.stSeqCtrlGeneral.eActiveSeqState := E_SEQ_GENERAL.EXECUTE;
	END_IF
  
END_IF

ELSE
  THIS^.stSeqCtrlGeneral.eActiveSeqState := E_SEQ_GENERAL.ERROR;
END_CASE
END_METHOD

METHOD PRIVATE _m_Seq_TO_WP1 : BOOL
VAR
  ActiveSeq: STRING;
END_VAR
//THIS^._m_GeneralStepSetting(StepType:=E_STEP_STATE_TYPE.INIT,
ActiveSeq := TO_STRING(THIS^.eSeq);

CASE THIS^.stSeqCtrlGeneral.eActiveSeqState OF
E_SEQ_GENERAL.READY:;

	
E_SEQ_GENERAL.EXECUTE:;
	IF TRUE
	THEN
		THIS^.stSeqCtrlGeneral.eActiveSeqState := E_SEQ_GENERAL.RESET;
	END_IF
  
E_SEQ_GENERAL.RESET:;
	stSeqCtrlGeneral.iInternalSeqStateCase := 0;
	IF TRUE
	THEN
		THIS^.stSeqCtrlGeneral.eActiveSeqState := E_SEQ_GENERAL.BUSY;
	END_IF
  
E_SEQ_GENERAL.BUSY:;
	CASE THIS^.stSeqCtrlGeneral.iInternalSeqStateCase OF
    0:  // Reset valve
      IF TRUE 
			THEN 
        itfSwitchToWP1.M_Set();
        itfSwitchToWP2.M_Reset();
        IF _m_Delay(tDelay) THEN
          THIS^.stSeqCtrlGeneral.iInternalSeqStateCase := 1000;
				END_IF
			END_IF
      
	ELSE
		THIS^.stSeqCtrlGeneral.eActiveSeqState := E_SEQ_GENERAL.DONE;  
	END_CASE
	THIS^.stSeqCtrlGeneral.strExtraInfo := CONCAT('Internal state: ', TO_STRING(THIS^.stSeqCtrlGeneral.iInternalSeqStateCase));

E_SEQ_GENERAL.DONE:;

E_SEQ_GENERAL.ERROR:;

E_SEQ_GENERAL.TIME_OUT:; 
IF TRUE
AND THIS^.stSeqCtrlGeneral.bTimeOutActiveQuit 
THEN
  THIS^.stSeqCtrlGeneral.strExtraInfo := 'Bitte quittieren und erneut testen';
  IF TRUE
  //AND itfOpMode.P_QUIT
  THEN
    THIS^.stSeqCtrlGeneral.eActiveSeqState := E_SEQ_GENERAL.EXECUTE;
	END_IF
  
END_IF

ELSE
  THIS^.stSeqCtrlGeneral.eActiveSeqState := E_SEQ_GENERAL.ERROR;
END_CASE
END_METHOD

METHOD PRIVATE _m_Seq_TO_WP2 : BOOL
VAR
  ActiveSeq: STRING;
END_VAR
//THIS^._m_GeneralStepSetting(StepType:=E_STEP_STATE_TYPE.INIT,
ActiveSeq := TO_STRING(THIS^.eSeq);

CASE THIS^.stSeqCtrlGeneral.eActiveSeqState OF
E_SEQ_GENERAL.READY:;

	
E_SEQ_GENERAL.EXECUTE:;
	IF TRUE
	THEN
		THIS^.stSeqCtrlGeneral.eActiveSeqState := E_SEQ_GENERAL.RESET;
	END_IF
  
E_SEQ_GENERAL.RESET:;
	stSeqCtrlGeneral.iInternalSeqStateCase := 0;
	IF TRUE
	THEN
		THIS^.stSeqCtrlGeneral.eActiveSeqState := E_SEQ_GENERAL.BUSY;
	END_IF
  
E_SEQ_GENERAL.BUSY:;
	CASE THIS^.stSeqCtrlGeneral.iInternalSeqStateCase OF
    0:  // Reset valve
      IF TRUE
			THEN 
        itfSwitchToWP1.M_Reset();
        itfSwitchToWP2.M_Set();
        IF _m_Delay(tDelay) THEN
          THIS^.stSeqCtrlGeneral.iInternalSeqStateCase := 1000;
				END_IF
			END_IF
      
	ELSE
		THIS^.stSeqCtrlGeneral.eActiveSeqState := E_SEQ_GENERAL.DONE;  
	END_CASE
	THIS^.stSeqCtrlGeneral.strExtraInfo := CONCAT('Internal state: ', TO_STRING(THIS^.stSeqCtrlGeneral.iInternalSeqStateCase));

E_SEQ_GENERAL.DONE:;

E_SEQ_GENERAL.ERROR:;

E_SEQ_GENERAL.TIME_OUT:; 
IF TRUE
AND THIS^.stSeqCtrlGeneral.bTimeOutActiveQuit 
THEN
  THIS^.stSeqCtrlGeneral.strExtraInfo := 'Bitte quittieren und erneut testen';
  IF TRUE
  //AND itfOpMode.P_QUIT
  THEN
    THIS^.stSeqCtrlGeneral.eActiveSeqState := E_SEQ_GENERAL.EXECUTE;
	END_IF
  
END_IF

ELSE
  THIS^.stSeqCtrlGeneral.eActiveSeqState := E_SEQ_GENERAL.ERROR;
END_CASE
END_METHOD

METHOD PRIVATE _m_SequenceManager
VAR_INPUT
END_VAR
IF FALSE
//AND THIS^.eActiveSeqState=DONE 
AND eLastSeq<>eSeq
THEN
	IF THIS^.stSeqCtrlGeneral.eActiveSeqState<>E_SEQ_GENERAL.EXECUTE THEN
		THIS^.stSeqCtrlGeneral.eActiveSeqState:=E_SEQ_GENERAL.READY;
	END_IF
END_IF

eSeq := eNextSeq;

//DelayTimer und TimeOut Timer verwalten
stSeqCtrlGeneral.bActiveStep:=	TRUE
				AND eLastSeq					=	eSeq
				AND stSeqCtrlGeneral.eLastActiveSeqState			=	stSeqCtrlGeneral.eActiveSeqState
				AND	stSeqCtrlGeneral.iLastInternalSeqStateCase	=	stSeqCtrlGeneral.iInternalSeqStateCase
				;
			
IF NOT stSeqCtrlGeneral.bActiveStep THEN
	stSeqCtrlGeneral.bDelayActive:=FALSE;
	stSeqCtrlGeneral.bTimeOutActiveQuit:=FALSE;
	stSeqCtrlGeneral.bTimeOutActiveNoQuit:=FALSE;
  THIS^.stSeqCtrlGeneral.strExtraInfo:='';
END_IF

_m_SaveLastStep();
stSeqCtrlGeneral.tonDelay	(IN:=stSeqCtrlGeneral.bActiveStep AND stSeqCtrlGeneral.bDelayActive, 		PT:=stSeqCtrlGeneral.tDelay);
stSeqCtrlGeneral.tonTimeOut	(IN:=stSeqCtrlGeneral.bActiveStep AND (stSeqCtrlGeneral.bTimeOutActiveNoQuit OR stSeqCtrlGeneral.bTimeOutActiveQuit), 	PT:=stSeqCtrlGeneral.tTimeOut);
stSeqCtrlGeneral.tonStepTime	(IN:= stSeqCtrlGeneral.bActiveStep, PT:= T#24H);

IF stSeqCtrlGeneral.tonTimeOut.Q  THEN
	stSeqCtrlGeneral.eActiveSeqState:=E_SEQ_GENERAL.TIME_OUT;
END_IF

IF stSeqCtrlGeneral.iError<>0 THEN
	eSeq:=E_SEQ_VALVE.ERROR_SEQ;
END_IF



eLastSeq					:=	eSeq;
stSeqCtrlGeneral.eLastActiveSeqState			:=	stSeqCtrlGeneral.eActiveSeqState;
stSeqCtrlGeneral.iLastInternalSeqStateCase	:=	stSeqCtrlGeneral.iInternalSeqStateCase;

// Reset set ready state
IF THIS^.stSeqCtrlGeneral.bExitSetReadyState THEN
  THIS^.stSeqCtrlGeneral.bExitSetReadyState := FALSE;
END_IF
END_METHOD

METHOD PRIVATE _m_TimeOut : BOOL
VAR_INPUT
	bTimeoutActiveToQuit:	BOOL;
	bTimeOutActiveNoQuit:	BOOL;
	tTimeOut:				TIME;	
END_VAR
THIS^.stSeqCtrlGeneral.bTimeOutActiveQuit:=	bTimeoutActiveToQuit;
THIS^.stSeqCtrlGeneral.bTimeOutActiveNoQuit:=	bTimeOutActiveNoQuit;
THIS^.stSeqCtrlGeneral.tTimeOut:=			tTimeOut;
_m_TimeOut:=FALSE;
IF THIS^.stSeqCtrlGeneral.tonTimeOut.Q THEN
	_m_TimeOut:=TRUE;
END_IF
END_METHOD

METHOD FB_init : BOOL
VAR_INPUT
	bInitRetains : BOOL; // if TRUE, the retain variables are initialized (warm start / cold start)
	bInCopyCode : BOOL;  // if TRUE, the instance afterwards gets moved into the copy code (online change)
  
  itfOpMode:											                        I_OP_MODE;
  itfEventLogger:                                         I_EVENT_LOGGER;
  itfSwitchToWP1:                                         I_BINARY_OUTPUT;
  itfSwitchToWP2:                                         I_BINARY_OUTPUT;
END_VAR
THIS^.itfOpMode := itfOpMode;
THIS^.itfEventLogger := itfEventLogger;
THIS^.itfSwitchToWP1 := itfSwitchToWP1;
THIS^.itfSwitchToWP2 := itfSwitchToWP2;
END_METHOD

METHOD M_Reset : BOOL
VAR_INPUT
END_VAR
M_Reset := THIS^.stSeqCtrlGeneral.eActiveSeqState = E_SEQ_GENERAL.DONE;

// Assign input

// General
IF THIS^.stSeqCtrlGeneral.eActiveSeqState = E_SEQ_GENERAL.READY THEN
  THIS^.eNextSeq := E_SEQ_VALVE.INIT;
  THIS^.stSeqCtrlGeneral.eActiveSeqState := E_SEQ_GENERAL.EXECUTE;
END_IF
END_METHOD

(*=== Method: M_Run  ============================================

 @brief: Here is the global code (Timer, Event, Flange,...)*)
METHOD M_Run
END_METHOD

METHOD M_SetReady : BOOL
VAR_INPUT
END_VAR
M_SetReady := TRUE
              AND THIS^.stSeqCtrlGeneral.eActiveSeqState = E_SEQ_GENERAL.READY
              AND THIS^.eSeq = E_SEQ_VALVE.BASE;

THIS^.stSeqCtrlGeneral.eActiveSeqState := E_SEQ_GENERAL.READY;
THIS^.eNextSeq := E_SEQ_VALVE.BASE;
END_METHOD

METHOD M_ToHP : BOOL
VAR_INPUT
  tDelay:         TIME;
END_VAR
M_ToHP := THIS^.stSeqCtrlGeneral.eActiveSeqState = E_SEQ_GENERAL.DONE;

// Assign input
THIS^.tDelay := tDelay;

// General
IF THIS^.stSeqCtrlGeneral.eActiveSeqState = E_SEQ_GENERAL.READY THEN
  THIS^.eNextSeq := E_SEQ_VALVE.SET_HP;
  THIS^.stSeqCtrlGeneral.eActiveSeqState := E_SEQ_GENERAL.EXECUTE;
END_IF
END_METHOD

METHOD M_ToWP1 : BOOL
VAR_INPUT
  tDelay:        TIME;
END_VAR
M_ToWP1 := THIS^.stSeqCtrlGeneral.eActiveSeqState = E_SEQ_GENERAL.DONE;

// Assign input
THIS^.tDelay := tDelay;

// General
IF THIS^.stSeqCtrlGeneral.eActiveSeqState = E_SEQ_GENERAL.READY THEN
  THIS^.eNextSeq := E_SEQ_VALVE.SET_WP1;
  THIS^.stSeqCtrlGeneral.eActiveSeqState := E_SEQ_GENERAL.EXECUTE;
END_IF
END_METHOD

METHOD M_ToWP2 : BOOL
VAR_INPUT
  tDelay:        TIME;
END_VAR
M_ToWP2 := THIS^.stSeqCtrlGeneral.eActiveSeqState = E_SEQ_GENERAL.DONE;

// Assign input
THIS^.tDelay := tDelay;

// General
IF THIS^.stSeqCtrlGeneral.eActiveSeqState = E_SEQ_GENERAL.READY THEN
  THIS^.eNextSeq := E_SEQ_VALVE.SET_WP2;
  THIS^.stSeqCtrlGeneral.eActiveSeqState := E_SEQ_GENERAL.EXECUTE;
END_IF
END_METHOD

(*=== Property: P_Event  ============================================

 @param [set]: 	Set the Structure "ST_EVENT" from another Object
 @param [get]: 	Return the Structure "ST_EVENT", it contains the actual 
					event of the Object *)
PROPERTY P_Event : GenLib.ST_EVENT
GET
END_GET
SET
END_SET
END_PROPERTY

{warning 'Eigenschaftenimplementierung hinzufügen'}
(*=== Property: P_FullObjectPath  ============================================

 @param [set]: 	Set the Object Path (Clear String of Object)
 @param [get]: 	Return the Objectpath *)
PROPERTY P_FullObjectPath : STRING
GET
END_GET
SET
END_SET
END_PROPERTY

{warning 'Eigenschaftenimplementierung hinzufügen'}
(*=== Property: P_Global_Ack  ============================================

 @param [set]: 	Set the Bit for Ack from another Object
 @param [get]: 	Return the state of Ack Bit*)
PROPERTY P_Global_Ack : BOOL
GET
END_GET
SET
END_SET
END_PROPERTY

{warning 'Eigenschaftenimplementierung hinzufügen'}
(*=== Property: P_GlobalID  ============================================

 @param [set]: 	-
 @param [get]: 	Return the string of instance path*)
PROPERTY P_GlobalID : STRING
GET
END_GET
END_PROPERTY

PROPERTY P_InHP : BOOL
GET
P_InHP := NOT THIS^.itfSwitchToWP1.P_State AND NOT THIS^.itfSwitchToWP2.P_State;
END_GET
END_PROPERTY

PROPERTY P_InWP1 : BOOL
GET
P_InWP1 := THIS^.itfSwitchToWP1.P_State AND NOT THIS^.itfSwitchToWP2.P_State;
END_GET
END_PROPERTY

{warning 'Eigenschaftenimplementierung hinzufügen'}
PROPERTY P_InWP2 : BOOL
GET
P_InWP2 := NOT THIS^.itfSwitchToWP1.P_State AND THIS^.itfSwitchToWP2.P_State;
END_GET
END_PROPERTY

{warning 'Eigenschaftenimplementierung hinzufügen'}
PROPERTY P_ReadyState : BOOL
GET
P_ReadyState := THIS^.stSeqCtrlGeneral.eActiveSeqState = E_SEQ_GENERAL.READY;
END_GET
END_PROPERTY

END_FUNCTION_BLOCK

// ---- MODULE/ACTOR_VALVE/VALVE/POU/FB_PRV_PROP.TcPOU
FUNCTION_BLOCK FB_PRV_PROP IMPLEMENTS I_PRV_PROP
VAR //General
	{attribute 'instance-path'} 
  {attribute 'noinit'} 
	strInstancePath:									                      STRING;
	bInit: 												                          BOOL:=TRUE;
	strFullObjectPath: 								                      STRING;
	stEvent:											                          ST_EVENT;
	bAck:												                            BOOL;
	
END_VAR
VAR   // From FB_init	
	itfOpMode:											                        I_OP_MODE; 
  itfEventLogger:                                         I_EVENT_LOGGER;
  rMaxLimitInBar:                                         REAL;
END_VAR                                      				
VAR	// Step chain control                				
  eSeq, eLastSeq, eNextSeq:					                      E_SEQ_VALVE; 
                  				
  //eActiveSeqState, eLastActiveSeqState:                 E_SEQ_GENERAL;
	(*
  iInternalSeqStateCase, iLastInternalSeqStateCase:       INT:=0;       
	tonDelay, tonTimeOut, tonStepTime:						          TON;
	tDelay:													                        TIME := T#100MS;
	tTimeOut:												                        TIME := T#100MS;
	tTimeOutExt:											                      TIME := T#100MS;
	bDelayActive, bTimeOutActiveQuit, bTimeOutActiveNoQuit:	BOOL;//Timer Option
	bActiveStep, bDebugAcitve, bDebugNext:					        BOOL;//Debug Option
	i:														                          INT;
 	iError:													                        INT; //ERROR-CODE                    	                   		
	listLastSteps:											                    ARRAY[0..49] OF ST_LAST_STEPS;	
	strExtraInfo:											                      STRING; 
	eStep_Type:												                      E_STEP_STATE_TYPE; 
	bDebugModeActive:										                    BOOL;   
	bWaitForBreakpoint:										                  BOOL;
	bBreakpointActive:										                  BOOL;
	bDebugResume:											                      BOOL;   
	listBreakpoint:											                    ARRAY[0..10] OF  INT;    
*)
i:														                            INT;
stSeqCtrlGeneral:											                    ST_SEQ_CTRL_GEN;     	
END_VAR                                             		
VAR                                                 		
	bMethodeFromExtStarted:									                BOOL;
	bMethodeFromExtActive:									                BOOL;
	bMethodeFromExtDone:									                  BOOL;
	strTemp:												                        STRING;
END_VAR   
VAR
  stHMI:                                                  ST_HMI_VALVE;
  rLimit:                                                 REAL;
  // For property
  rLimitInPercent:                                        REAL;
  rLimitInBar:                                            REAL;
  ePressureType:                                          E_PRESSURE_TYPE;
END_VAR                  	
VAR_TEMP                    	
	iTemp:										                              INT;
END_VAR
VAR_OUTPUT
  iTargetVal:                                             INT;
END_VAR

// Set FBs and Interfaces ready after switch internal step
IF stSeqCtrlGeneral.iInternalSeqStateCase <> stSeqCtrlGeneral.iLastInternalSeqStateCase AND NOT stSeqCtrlGeneral.bExitSetReadyState THEN
  IF TRUE
  //AND ...
  THEN
    stSeqCtrlGeneral.bExitSetReadyState := TRUE;
  ELSE
    RETURN;
  END_IF
END_IF

stSeqCtrlGeneral.strObject := F_CreateObjectName(strInstancePath);

// First method call
_m_SequenceManager();
//_m_SaveLastStep();

CASE eSeq OF 
  E_SEQ_VALVE.BASE:;
  
	E_SEQ_VALVE.INIT: _m_Seq_INIT();
		IF TRUE
		AND (stSeqCtrlGeneral.eActiveSeqState = E_SEQ_GENERAL.DONE) 
		THEN
			eSeq := E_SEQ_VALVE.BASE;
		END_IF
		
	E_SEQ_VALVE.SETUP:;
  
	// Process
  E_SEQ_VALVE.SET_LIMIT: _m_Seq_SET_LIMIT();
    IF TRUE
		AND (stSeqCtrlGeneral.eActiveSeqState = E_SEQ_GENERAL.DONE) 
		THEN
			eSeq := E_SEQ_VALVE.BASE;
		END_IF

  // End
	E_SEQ_VALVE.END:;
	E_SEQ_VALVE.ERROR_SEQ:;	
END_CASE

strTemp:=TO_STRING(eSeq);

METHOD PRIVATE _m_DebugManager
VAR_INPUT
	iStepID: int;
END_VAR
IF TRUE
AND THIS^.stSeqCtrlGeneral.bDebugModeActive 
AND NOT THIS^.stSeqCtrlGeneral.bActiveStep
THEN


THIS^.stSeqCtrlGeneral.bBreakpointActive:=FALSE;

FOR i:=0 TO 10 DO
	
	IF TRUE
	AND iStepID=THIS^.stSeqCtrlGeneral.listBreakpoint[i] 
	AND iStepID<>0
	THEN
		EXIT;
	END_IF
END_FOR
IF (i<=10) THEN
	THIS^.stSeqCtrlGeneral.bBreakpointActive:=TRUE;
END_IF

END_IF
END_METHOD

METHOD PRIVATE _m_Delay : BOOL
VAR_INPUT
	DelayTime:	TIME;
END_VAR
THIS^.stSeqCtrlGeneral.bDelayActive:=TRUE;
THIS^.stSeqCtrlGeneral.tDelay:=DelayTime;
_m_Delay:=FALSE;
IF THIS^.stSeqCtrlGeneral.tonDelay.Q THEN
	_m_Delay:=TRUE;
END_IF
END_METHOD

METHOD PRIVATE _m_GeneralStepSetting : BOOL
VAR_INPUT
	StepType:			    	E_STEP_STATE_TYPE;
	InfoTextID:					STRING(20);
	EnableDebug:	   			BOOL;	
	
END_VAR
IF THIS^.stSeqCtrlGeneral.bActiveStep THEN
	THIS^.stSeqCtrlGeneral.eStep_Type:=StepType;
	THIS^.stSeqCtrlGeneral.strExtraInfo:= GenLib.F_RET_TXTLIST_ENTRY(strPortNr:='851',strID:='',strTxtLstName:=InfoTextID);
END_IF
END_METHOD

METHOD PRIVATE _m_SaveLastStep : BOOL
VAR_INPUT
END_VAR
VAR
	i: dint;
END_VAR
IF NOT THIS^.stSeqCtrlGeneral.bActiveStep THEN
	
	FOR i:=49 TO 1 BY -1 DO
			stSeqCtrlGeneral.listLastSteps[i].strStepName:=stSeqCtrlGeneral.listLastSteps[i-1].strStepName;
			stSeqCtrlGeneral.listLastSteps[i].tStepTime:=stSeqCtrlGeneral.listLastSteps[i-1].tStepTime;
			stSeqCtrlGeneral.listLastSteps[i].tDelayTime:=stSeqCtrlGeneral.listLastSteps[i-1].tDelayTime;
	END_FOR
	stSeqCtrlGeneral.listLastSteps[0].strStepName:=TO_STRING(THIS^.eSeq);
	stSeqCtrlGeneral.listLastSteps[1].tStepTime:=THIS^.stSeqCtrlGeneral.tonStepTime.ET;
	stSeqCtrlGeneral.listLastSteps[1].tStepTime:=THIS^.stSeqCtrlGeneral.tonDelay.ET;
ELSE
	stSeqCtrlGeneral.listLastSteps[0].tStepTime:=THIS^.stSeqCtrlGeneral.tonStepTime.ET;
	stSeqCtrlGeneral.listLastSteps[0].tDelayTime:=THIS^.stSeqCtrlGeneral.tonDelay.ET;	
END_IF
END_METHOD

METHOD PRIVATE _m_Seq_INIT : BOOL
VAR
  ActiveSeq: STRING;
END_VAR
//THIS^._m_GeneralStepSetting(StepType:=E_STEP_STATE_TYPE.INIT,
ActiveSeq := TO_STRING(THIS^.eSeq);

CASE THIS^.stSeqCtrlGeneral.eActiveSeqState OF
E_SEQ_GENERAL.READY:;

	
E_SEQ_GENERAL.EXECUTE:;
	IF TRUE
	THEN
		THIS^.stSeqCtrlGeneral.eActiveSeqState := E_SEQ_GENERAL.RESET;
	END_IF
  
E_SEQ_GENERAL.RESET:;
	stSeqCtrlGeneral.iInternalSeqStateCase := 0;
	IF TRUE
	THEN
		THIS^.stSeqCtrlGeneral.eActiveSeqState := E_SEQ_GENERAL.BUSY;
	END_IF
  
E_SEQ_GENERAL.BUSY:;
	CASE THIS^.stSeqCtrlGeneral.iInternalSeqStateCase OF
    0:  // Reset valve
      IF TRUE 
			THEN 
        THIS^.iTargetVal := 0;
        THIS^.stSeqCtrlGeneral.iInternalSeqStateCase := 1000;
			END_IF
      
	ELSE
		THIS^.stSeqCtrlGeneral.eActiveSeqState := E_SEQ_GENERAL.DONE;  
	END_CASE
	THIS^.stSeqCtrlGeneral.strExtraInfo := CONCAT('Internal state: ', TO_STRING(THIS^.stSeqCtrlGeneral.iInternalSeqStateCase));

E_SEQ_GENERAL.DONE:;

E_SEQ_GENERAL.ERROR:;

E_SEQ_GENERAL.TIME_OUT:; 
IF TRUE
AND THIS^.stSeqCtrlGeneral.bTimeOutActiveQuit 
THEN
  THIS^.stSeqCtrlGeneral.strExtraInfo := 'Bitte quittieren und erneut testen';
  IF TRUE
  //AND itfOpMode.P_QUIT
  THEN
    THIS^.stSeqCtrlGeneral.eActiveSeqState := E_SEQ_GENERAL.EXECUTE;
	END_IF
  
END_IF

ELSE
  THIS^.stSeqCtrlGeneral.eActiveSeqState := E_SEQ_GENERAL.ERROR;
END_CASE
END_METHOD

METHOD PRIVATE _m_Seq_SET_LIMIT : BOOL
VAR
  ActiveSeq:  STRING;
  iTmp:       INT;
END_VAR
//THIS^._m_GeneralStepSetting(StepType:=E_STEP_STATE_TYPE.INIT,
ActiveSeq := TO_STRING(THIS^.eSeq);

CASE THIS^.stSeqCtrlGeneral.eActiveSeqState OF
E_SEQ_GENERAL.READY:;

	
E_SEQ_GENERAL.EXECUTE:;
	IF TRUE
	THEN
		THIS^.stSeqCtrlGeneral.eActiveSeqState := E_SEQ_GENERAL.RESET;
	END_IF
  
E_SEQ_GENERAL.RESET:;
	stSeqCtrlGeneral.iInternalSeqStateCase := 0;
	IF TRUE
	THEN
		THIS^.stSeqCtrlGeneral.eActiveSeqState := E_SEQ_GENERAL.BUSY;
	END_IF
  
E_SEQ_GENERAL.BUSY:;
	CASE THIS^.stSeqCtrlGeneral.iInternalSeqStateCase OF
    0:  // Set valve
      IF TRUE 
			THEN 
        IF THIS^.ePressureType = E_PRESSURE_TYPE.VALUE THEN
          THIS^.iTargetVal := TO_INT(THIS^.rLimit);
        ELSE
          iTmp := TO_INT(327.67 * THIS^.rLimitInPercent);
          IF iTmp < 0 THEN 
            iTmp := iTmp - 1;
          END_IF
          THIS^.iTargetVal := iTmp;
        END_IF
        THIS^.stSeqCtrlGeneral.iInternalSeqStateCase := 1000;
			END_IF
      
	ELSE
		THIS^.stSeqCtrlGeneral.eActiveSeqState := E_SEQ_GENERAL.DONE;  
	END_CASE
	THIS^.stSeqCtrlGeneral.strExtraInfo := CONCAT('Internal state: ', TO_STRING(THIS^.stSeqCtrlGeneral.iInternalSeqStateCase));

E_SEQ_GENERAL.DONE:;

E_SEQ_GENERAL.ERROR:;

E_SEQ_GENERAL.TIME_OUT:; 
IF TRUE
AND THIS^.stSeqCtrlGeneral.bTimeOutActiveQuit 
THEN
  THIS^.stSeqCtrlGeneral.strExtraInfo := 'Bitte quittieren und erneut testen';
  IF TRUE
  //AND itfOpMode.P_QUIT
  THEN
    THIS^.stSeqCtrlGeneral.eActiveSeqState := E_SEQ_GENERAL.EXECUTE;
	END_IF
  
END_IF

ELSE
  THIS^.stSeqCtrlGeneral.eActiveSeqState := E_SEQ_GENERAL.ERROR;
END_CASE
END_METHOD

METHOD PRIVATE _m_SequenceManager
VAR_INPUT
END_VAR
IF FALSE
//AND THIS^.eActiveSeqState=DONE 
AND eLastSeq<>eSeq
THEN
	IF THIS^.stSeqCtrlGeneral.eActiveSeqState<>E_SEQ_GENERAL.EXECUTE THEN
		THIS^.stSeqCtrlGeneral.eActiveSeqState:=E_SEQ_GENERAL.READY;
	END_IF
END_IF

eSeq := eNextSeq;

//DelayTimer und TimeOut Timer verwalten
stSeqCtrlGeneral.bActiveStep:=	TRUE
				AND eLastSeq					=	eSeq
				AND stSeqCtrlGeneral.eLastActiveSeqState			=	stSeqCtrlGeneral.eActiveSeqState
				AND	stSeqCtrlGeneral.iLastInternalSeqStateCase	=	stSeqCtrlGeneral.iInternalSeqStateCase
				;
			
IF NOT stSeqCtrlGeneral.bActiveStep THEN
	stSeqCtrlGeneral.bDelayActive:=FALSE;
	stSeqCtrlGeneral.bTimeOutActiveQuit:=FALSE;
	stSeqCtrlGeneral.bTimeOutActiveNoQuit:=FALSE;
  THIS^.stSeqCtrlGeneral.strExtraInfo:='';
END_IF

_m_SaveLastStep();
stSeqCtrlGeneral.tonDelay	(IN:=stSeqCtrlGeneral.bActiveStep AND stSeqCtrlGeneral.bDelayActive, 		PT:=stSeqCtrlGeneral.tDelay);
stSeqCtrlGeneral.tonTimeOut	(IN:=stSeqCtrlGeneral.bActiveStep AND (stSeqCtrlGeneral.bTimeOutActiveNoQuit OR stSeqCtrlGeneral.bTimeOutActiveQuit), 	PT:=stSeqCtrlGeneral.tTimeOut);
stSeqCtrlGeneral.tonStepTime	(IN:= stSeqCtrlGeneral.bActiveStep, PT:= T#24H);

IF stSeqCtrlGeneral.tonTimeOut.Q  THEN
	stSeqCtrlGeneral.eActiveSeqState:=E_SEQ_GENERAL.TIME_OUT;
END_IF

IF stSeqCtrlGeneral.iError<>0 THEN
	eSeq:=E_SEQ_VALVE.ERROR_SEQ;
END_IF



eLastSeq					:=	eSeq;
stSeqCtrlGeneral.eLastActiveSeqState			:=	stSeqCtrlGeneral.eActiveSeqState;
stSeqCtrlGeneral.iLastInternalSeqStateCase	:=	stSeqCtrlGeneral.iInternalSeqStateCase;

// Reset set ready state
IF THIS^.stSeqCtrlGeneral.bExitSetReadyState THEN
  THIS^.stSeqCtrlGeneral.bExitSetReadyState := FALSE;
END_IF
END_METHOD

METHOD PRIVATE _m_TimeOut : BOOL
VAR_INPUT
	bTimeoutActiveToQuit:	BOOL;
	bTimeOutActiveNoQuit:	BOOL;
	tTimeOut:				TIME;	
END_VAR
THIS^.stSeqCtrlGeneral.bTimeOutActiveQuit:=	bTimeoutActiveToQuit;
THIS^.stSeqCtrlGeneral.bTimeOutActiveNoQuit:=	bTimeOutActiveNoQuit;
THIS^.stSeqCtrlGeneral.tTimeOut:=			tTimeOut;
_m_TimeOut:=FALSE;
IF THIS^.stSeqCtrlGeneral.tonTimeOut.Q THEN
	_m_TimeOut:=TRUE;
END_IF
END_METHOD

METHOD FB_init : BOOL
VAR_INPUT
	bInitRetains : BOOL; // if TRUE, the retain variables are initialized (warm start / cold start)
	bInCopyCode : BOOL;  // if TRUE, the instance afterwards gets moved into the copy code (online change)
  
  itfOpMode:											                        I_OP_MODE; 
  itfEventLogger:                                         I_EVENT_LOGGER;
  rMaxLimitInBar:                                         REAL;
END_VAR
THIS^.itfOpMode := itfOpMode;
THIS^.itfEventLogger := itfEventLogger;
THIS^.rMaxLimitInBar := rMaxLimitInBar;
END_METHOD

METHOD M_Reset : BOOL
VAR_INPUT
END_VAR
M_Reset := THIS^.stSeqCtrlGeneral.eActiveSeqState = E_SEQ_GENERAL.DONE;

// Assign input

// General
IF THIS^.stSeqCtrlGeneral.eActiveSeqState = E_SEQ_GENERAL.READY THEN
  THIS^.eNextSeq := E_SEQ_VALVE.INIT;
  THIS^.stSeqCtrlGeneral.eActiveSeqState := E_SEQ_GENERAL.EXECUTE;
END_IF
END_METHOD

{warning 'Methodenimplementierung hinzufügen'}
(*=== Method: M_Run  ============================================

 @brief: Here is the global code (Timer, Event, Flange,...)*)
METHOD M_Run
END_METHOD

METHOD M_SetLimit : BOOL
VAR_INPUT
  ePressureType:      E_PRESSURE_TYPE;
  rLimit:             REAL;
END_VAR
M_SetLimit := THIS^.stSeqCtrlGeneral.eActiveSeqState = E_SEQ_GENERAL.DONE;

// Assign input
THIS^.ePressureType := ePressureType;
IF ePressureType = E_PRESSURE_TYPE.PERCENT THEN
  IF ABS(rLimit) > 100 THEN
    rLimit := 100;
	END_IF
  THIS^.rLimit := ABS(rLimit);
  THIS^.rLimitInPercent := THIS^.rLimit;
  // Calc value in bar
  THIS^.rLimitInBar := THIS^.rMaxLimitInBar * THIS^.rLimitInPercent / 100;
ELSIF ePressureType = E_PRESSURE_TYPE.BAR THEN
  IF ABS(rLimit) > THIS^.rMaxLimitInBar THEN
    rLimit := THIS^.rMaxLimitInBar;
	END_IF
  THIS^.rLimit := rLimit;
  THIS^.rLimitInBar := rLimit;
  // Calc value in percent
  THIS^.rLimitInPercent := 100 / THIS^.rMaxLimitInBar * THIS^.rLimitInBar;
ELSE
  THIS^.rLimit := rLimit;
END_IF

// General
IF THIS^.stSeqCtrlGeneral.eActiveSeqState = E_SEQ_GENERAL.READY THEN
  THIS^.eNextSeq := E_SEQ_VALVE.SET_LIMIT;
  THIS^.stSeqCtrlGeneral.eActiveSeqState := E_SEQ_GENERAL.EXECUTE;
END_IF
END_METHOD

METHOD M_SetReady : BOOL
VAR_INPUT
END_VAR
M_SetReady := TRUE
              AND THIS^.stSeqCtrlGeneral.eActiveSeqState = E_SEQ_GENERAL.READY
              AND THIS^.eSeq = E_SEQ_VALVE.BASE;

THIS^.stSeqCtrlGeneral.eActiveSeqState := E_SEQ_GENERAL.READY;
THIS^.eNextSeq := E_SEQ_VALVE.BASE;
END_METHOD

{warning 'Eigenschaftenimplementierung hinzufügen'}
(*=== Property: P_Event  ============================================

 @param [set]: 	Set the Structure "ST_EVENT" from another Object
 @param [get]: 	Return the Structure "ST_EVENT", it contains the actual 
					event of the Object *)
PROPERTY P_Event : GenLib.ST_EVENT
GET
END_GET
SET
END_SET
END_PROPERTY

{warning 'Eigenschaftenimplementierung hinzufügen'}
(*=== Property: P_FullObjectPath  ============================================

 @param [set]: 	Set the Object Path (Clear String of Object)
 @param [get]: 	Return the Objectpath *)
PROPERTY P_FullObjectPath : STRING
GET
END_GET
SET
END_SET
END_PROPERTY

{warning 'Eigenschaftenimplementierung hinzufügen'}
(*=== Property: P_Global_Ack  ============================================

 @param [set]: 	Set the Bit for Ack from another Object
 @param [get]: 	Return the state of Ack Bit*)
PROPERTY P_Global_Ack : BOOL
GET
END_GET
SET
END_SET
END_PROPERTY

{warning 'Eigenschaftenimplementierung hinzufügen'}
(*=== Property: P_GlobalID  ============================================

 @param [set]: 	-
 @param [get]: 	Return the string of instance path*)
PROPERTY P_GlobalID : STRING
GET
END_GET
END_PROPERTY

PROPERTY P_LimitInBar : REAL
GET
P_LimitInBar := THIS^.rLimitInBar;
END_GET
END_PROPERTY

PROPERTY P_LimitInPercent : REAL
GET
P_LimitInPercent := THIS^.rLimitInPercent;
END_GET
END_PROPERTY

{warning 'Eigenschaftenimplementierung hinzufügen'}
PROPERTY P_MaxLimitInBar : REAL
GET
P_MaxLimitInBar := THIS^.rMaxLimitInBar;
END_GET
END_PROPERTY

{warning 'Eigenschaftenimplementierung hinzufügen'}
PROPERTY P_ReadyState : BOOL
GET
P_ReadyState := THIS^.stSeqCtrlGeneral.eActiveSeqState = E_SEQ_GENERAL.READY;
END_GET
END_PROPERTY

END_FUNCTION_BLOCK

// ---- MODULE/ACTOR_VALVE/VALVE/POU/FB_VALVE_X_3_PROP.TcPOU
FUNCTION_BLOCK FB_VALVE_X_3_PROP IMPLEMENTS I_VALVE_X_3_PROP
VAR_OUTPUT
  iAnalogSwitch:                                          INT;
END_VAR
VAR //General
	{attribute 'instance-path'} 
  {attribute 'noinit'} 
	strInstancePath:									                      STRING;
	bInit: 												                          BOOL:=TRUE;
	strFullObjectPath: 								                      STRING;
	stEvent:											                          ST_EVENT;
	bAck:												                            BOOL;
END_VAR
VAR   // From FB_init	
	itfOpMode:											                        I_OP_MODE;
  itfEventLogger:                                         I_EVENT_LOGGER;
END_VAR                                      				
VAR	// Step chain control                				
  eSeq, eLastSeq, eNextSeq:					                      E_SEQ_VALVE; 
                  				
  //eActiveSeqState, eLastActiveSeqState:                 E_SEQ_GENERAL;
	(*
  iInternalSeqStateCase, iLastInternalSeqStateCase:       INT:=0;       
	tonDelay, tonTimeOut, tonStepTime:						          TON;
	tDelay:													                        TIME := T#100MS;
	tTimeOut:												                        TIME := T#100MS;
	tTimeOutExt:											                      TIME := T#100MS;
	bDelayActive, bTimeOutActiveQuit, bTimeOutActiveNoQuit:	BOOL;//Timer Option
	bActiveStep, bDebugAcitve, bDebugNext:					        BOOL;//Debug Option
	i:														                          INT;
 	iError:													                        INT; //ERROR-CODE                    	                   		
	listLastSteps:											                    ARRAY[0..49] OF ST_LAST_STEPS;	
	strExtraInfo:											                      STRING; 
	eStep_Type:												                      E_STEP_STATE_TYPE; 
	bDebugModeActive:										                    BOOL;   
	bWaitForBreakpoint:										                  BOOL;
	bBreakpointActive:										                  BOOL;
	bDebugResume:											                      BOOL;   
	listBreakpoint:											                    ARRAY[0..10] OF  INT;    
*)
i:														                            INT;
stSeqCtrlGeneral:											                    ST_SEQ_CTRL_GEN;     	
END_VAR                                             		
VAR                                                 		
	bMethodeFromExtStarted:									                BOOL;
	bMethodeFromExtActive:									                BOOL;
	bMethodeFromExtDone:									                  BOOL;
	strTemp:												                        STRING;
END_VAR   
VAR
  stHMI:                                                  ST_HMI_VALVE;
  tDelay:                                                 TIME;
  rSpeedInPercent:                                        REAL;
END_VAR
VAR
  iOutputVal:                                             INT; 
END_VAR                 	
VAR_TEMP                    	
	iTemp:										                              INT;
END_VAR

// Set FBs and Interfaces ready after switch internal step
IF stSeqCtrlGeneral.iInternalSeqStateCase <> stSeqCtrlGeneral.iLastInternalSeqStateCase AND NOT stSeqCtrlGeneral.bExitSetReadyState THEN
  IF TRUE
  //AND ...
  THEN
    stSeqCtrlGeneral.bExitSetReadyState := TRUE;
  ELSE
    RETURN;
  END_IF
END_IF

stSeqCtrlGeneral.strObject := F_CreateObjectName(strInstancePath);

// First method call
_m_SequenceManager();
//_m_SaveLastStep();

CASE eSeq OF 
  E_SEQ_VALVE.BASE:;
  
	E_SEQ_VALVE.INIT: _m_Seq_INIT();
		IF TRUE
		AND (stSeqCtrlGeneral.eActiveSeqState = E_SEQ_GENERAL.DONE) 
		THEN
			eSeq := E_SEQ_VALVE.BASE;
		END_IF
		
	E_SEQ_VALVE.SETUP:;
  
	// Process
  E_SEQ_VALVE.SET_LIMIT: _m_Seq_VALVE_CTRL();
    IF TRUE
		AND (stSeqCtrlGeneral.eActiveSeqState = E_SEQ_GENERAL.DONE) 
		THEN
			eSeq := E_SEQ_VALVE.BASE;
		END_IF
    
  E_SEQ_VALVE.SET_LIMIT_SMOOTH: _m_Seq_VALVE_CTRL_SMOOTH();
    IF TRUE
		AND (stSeqCtrlGeneral.eActiveSeqState = E_SEQ_GENERAL.DONE) 
		THEN
			eSeq := E_SEQ_VALVE.BASE;
		END_IF

  // End
	E_SEQ_VALVE.END:;
	E_SEQ_VALVE.ERROR_SEQ:;	
END_CASE

strTemp:=TO_STRING(eSeq);

METHOD PRIVATE _m_DebugManager
VAR_INPUT
	iStepID: int;
END_VAR
IF TRUE
AND THIS^.stSeqCtrlGeneral.bDebugModeActive 
AND NOT THIS^.stSeqCtrlGeneral.bActiveStep
THEN


THIS^.stSeqCtrlGeneral.bBreakpointActive:=FALSE;

FOR i:=0 TO 10 DO
	
	IF TRUE
	AND iStepID=THIS^.stSeqCtrlGeneral.listBreakpoint[i] 
	AND iStepID<>0
	THEN
		EXIT;
	END_IF
END_FOR
IF (i<=10) THEN
	THIS^.stSeqCtrlGeneral.bBreakpointActive:=TRUE;
END_IF

END_IF
END_METHOD

METHOD PRIVATE _m_Delay : BOOL
VAR_INPUT
	DelayTime:	TIME;
END_VAR
THIS^.stSeqCtrlGeneral.bDelayActive:=TRUE;
THIS^.stSeqCtrlGeneral.tDelay:=DelayTime;
_m_Delay:=FALSE;
IF THIS^.stSeqCtrlGeneral.tonDelay.Q THEN
	_m_Delay:=TRUE;
END_IF
END_METHOD

METHOD PRIVATE _m_GeneralStepSetting : BOOL
VAR_INPUT
	StepType:			    	E_STEP_STATE_TYPE;
	InfoTextID:					STRING(20);
	EnableDebug:	   			BOOL;	
	
END_VAR
IF THIS^.stSeqCtrlGeneral.bActiveStep THEN
	THIS^.stSeqCtrlGeneral.eStep_Type:=StepType;
	THIS^.stSeqCtrlGeneral.strExtraInfo:= GenLib.F_RET_TXTLIST_ENTRY(strPortNr:='851',strID:='',strTxtLstName:=InfoTextID);
END_IF
END_METHOD

METHOD PRIVATE _m_SaveLastStep : BOOL
VAR_INPUT
END_VAR
VAR
	i: dint;
END_VAR
IF NOT THIS^.stSeqCtrlGeneral.bActiveStep THEN
	
	FOR i:=49 TO 1 BY -1 DO
			stSeqCtrlGeneral.listLastSteps[i].strStepName:=stSeqCtrlGeneral.listLastSteps[i-1].strStepName;
			stSeqCtrlGeneral.listLastSteps[i].tStepTime:=stSeqCtrlGeneral.listLastSteps[i-1].tStepTime;
			stSeqCtrlGeneral.listLastSteps[i].tDelayTime:=stSeqCtrlGeneral.listLastSteps[i-1].tDelayTime;
	END_FOR
	stSeqCtrlGeneral.listLastSteps[0].strStepName:=TO_STRING(THIS^.eSeq);
	stSeqCtrlGeneral.listLastSteps[1].tStepTime:=THIS^.stSeqCtrlGeneral.tonStepTime.ET;
	stSeqCtrlGeneral.listLastSteps[1].tStepTime:=THIS^.stSeqCtrlGeneral.tonDelay.ET;
ELSE
	stSeqCtrlGeneral.listLastSteps[0].tStepTime:=THIS^.stSeqCtrlGeneral.tonStepTime.ET;
	stSeqCtrlGeneral.listLastSteps[0].tDelayTime:=THIS^.stSeqCtrlGeneral.tonDelay.ET;	
END_IF
END_METHOD

METHOD PRIVATE _m_Seq_INIT : BOOL
VAR
  ActiveSeq: STRING;
END_VAR
//THIS^._m_GeneralStepSetting(StepType:=E_STEP_STATE_TYPE.INIT,
ActiveSeq := TO_STRING(THIS^.eSeq);

CASE THIS^.stSeqCtrlGeneral.eActiveSeqState OF
E_SEQ_GENERAL.READY:;

	
E_SEQ_GENERAL.EXECUTE:;
	IF TRUE
	THEN
		THIS^.stSeqCtrlGeneral.eActiveSeqState := E_SEQ_GENERAL.RESET;
	END_IF
  
E_SEQ_GENERAL.RESET:;
	stSeqCtrlGeneral.iInternalSeqStateCase := 0;
	IF TRUE
	THEN
		THIS^.stSeqCtrlGeneral.eActiveSeqState := E_SEQ_GENERAL.BUSY;
	END_IF
  
E_SEQ_GENERAL.BUSY:;
	CASE THIS^.stSeqCtrlGeneral.iInternalSeqStateCase OF
    0:  // Reset valve
      IF TRUE 
			THEN 
        iAnalogSwitch := 0;
        IF _m_Delay(T#1S) THEN
          THIS^.stSeqCtrlGeneral.iInternalSeqStateCase := 1000;
				END_IF
			END_IF
      
	ELSE
		THIS^.stSeqCtrlGeneral.eActiveSeqState := E_SEQ_GENERAL.DONE;  
	END_CASE
	THIS^.stSeqCtrlGeneral.strExtraInfo := CONCAT('Internal state: ', TO_STRING(THIS^.stSeqCtrlGeneral.iInternalSeqStateCase));

E_SEQ_GENERAL.DONE:;

E_SEQ_GENERAL.ERROR:;

E_SEQ_GENERAL.TIME_OUT:; 
IF TRUE
AND THIS^.stSeqCtrlGeneral.bTimeOutActiveQuit 
THEN
  THIS^.stSeqCtrlGeneral.strExtraInfo := 'Bitte quittieren und erneut testen';
  IF TRUE
  //AND itfOpMode.P_QUIT
  THEN
    THIS^.stSeqCtrlGeneral.eActiveSeqState := E_SEQ_GENERAL.EXECUTE;
	END_IF
  
END_IF

ELSE
  THIS^.stSeqCtrlGeneral.eActiveSeqState := E_SEQ_GENERAL.ERROR;
END_CASE
END_METHOD

METHOD PRIVATE _m_Seq_VALVE_CTRL : BOOL
VAR
  ActiveSeq:  STRING;
END_VAR
//THIS^._m_GeneralStepSetting(StepType:=E_STEP_STATE_TYPE.INIT,
ActiveSeq := TO_STRING(THIS^.eSeq);

CASE THIS^.stSeqCtrlGeneral.eActiveSeqState OF
E_SEQ_GENERAL.READY:;

	
E_SEQ_GENERAL.EXECUTE:;
	IF TRUE
	THEN
		THIS^.stSeqCtrlGeneral.eActiveSeqState := E_SEQ_GENERAL.RESET;
	END_IF
  
E_SEQ_GENERAL.RESET:;
	stSeqCtrlGeneral.iInternalSeqStateCase := 0;
	IF TRUE
	THEN
		THIS^.stSeqCtrlGeneral.eActiveSeqState := E_SEQ_GENERAL.BUSY;
	END_IF
  
E_SEQ_GENERAL.BUSY:;
	CASE THIS^.stSeqCtrlGeneral.iInternalSeqStateCase OF
    0:  // Calc output value
      IF TRUE 
			THEN 
        THIS^.iOutputVal := TO_INT(327.67 * THIS^.rSpeedInPercent);
        IF THIS^.iOutputVal < 0 THEN 
          THIS^.iOutputVal := THIS^.iOutputVal - 1;
        END_IF
        iAnalogSwitch := THIS^.iOutputVal;
        THIS^.stSeqCtrlGeneral.iInternalSeqStateCase := 10;
			END_IF
      
    10:  // Set output value
      IF TRUE 
			THEN 
        iAnalogSwitch := THIS^.iOutputVal;
        THIS^.stSeqCtrlGeneral.iInternalSeqStateCase := 1000;
			END_IF
      
	ELSE
		THIS^.stSeqCtrlGeneral.eActiveSeqState := E_SEQ_GENERAL.DONE;  
	END_CASE
	THIS^.stSeqCtrlGeneral.strExtraInfo := CONCAT('Internal state: ', TO_STRING(THIS^.stSeqCtrlGeneral.iInternalSeqStateCase));

E_SEQ_GENERAL.DONE:;

E_SEQ_GENERAL.ERROR:;

E_SEQ_GENERAL.TIME_OUT:; 
IF TRUE
AND THIS^.stSeqCtrlGeneral.bTimeOutActiveQuit 
THEN
  THIS^.stSeqCtrlGeneral.strExtraInfo := 'Bitte quittieren und erneut testen';
  IF TRUE
  //AND itfOpMode.P_QUIT
  THEN
    THIS^.stSeqCtrlGeneral.eActiveSeqState := E_SEQ_GENERAL.EXECUTE;
	END_IF
  
END_IF

ELSE
  THIS^.stSeqCtrlGeneral.eActiveSeqState := E_SEQ_GENERAL.ERROR;
END_CASE
END_METHOD

METHOD PRIVATE _m_Seq_VALVE_CTRL_SMOOTH : BOOL
VAR
  ActiveSeq:  STRING;
END_VAR
//THIS^._m_GeneralStepSetting(StepType:=E_STEP_STATE_TYPE.INIT,
ActiveSeq := TO_STRING(THIS^.eSeq);

CASE THIS^.stSeqCtrlGeneral.eActiveSeqState OF
E_SEQ_GENERAL.READY:;

	
E_SEQ_GENERAL.EXECUTE:;
	IF TRUE
	THEN
		THIS^.stSeqCtrlGeneral.eActiveSeqState := E_SEQ_GENERAL.RESET;
	END_IF
  
E_SEQ_GENERAL.RESET:;
	stSeqCtrlGeneral.iInternalSeqStateCase := 0;
	IF TRUE
	THEN
		THIS^.stSeqCtrlGeneral.eActiveSeqState := E_SEQ_GENERAL.BUSY;
	END_IF
  
E_SEQ_GENERAL.BUSY:;
	CASE THIS^.stSeqCtrlGeneral.iInternalSeqStateCase OF
    0:  // Calc output value
      IF TRUE 
			THEN 
        THIS^.iOutputVal := TO_INT(327.67 * THIS^.rSpeedInPercent);
        IF THIS^.iOutputVal < 0 THEN 
          THIS^.iOutputVal := THIS^.iOutputVal - 1;
        END_IF
        iAnalogSwitch := THIS^.iOutputVal;
        THIS^.stSeqCtrlGeneral.iInternalSeqStateCase := 10;
			END_IF
      
    10:  // Set output value
      IF TRUE 
			THEN 
        IF iAnalogSwitch > THIS^.iOutputVal + 100 THEN
          iAnalogSwitch := iAnalogSwitch - 100;
        ELSIF iAnalogSwitch < THIS^.iOutputVal - 100 THEN
          iAnalogSwitch := iAnalogSwitch + 100;
        END_IF
        IF ABS(iAnalogSwitch - THIS^.iOutputVal) <= 100 THEN
          THIS^.stSeqCtrlGeneral.iInternalSeqStateCase := 20;
        END_IF
			END_IF
      
    20:  // Set output value
      IF TRUE 
			THEN 
        iAnalogSwitch := THIS^.iOutputVal;
        THIS^.stSeqCtrlGeneral.iInternalSeqStateCase := 1000;
			END_IF
      
	ELSE
		THIS^.stSeqCtrlGeneral.eActiveSeqState := E_SEQ_GENERAL.DONE;  
	END_CASE
	THIS^.stSeqCtrlGeneral.strExtraInfo := CONCAT('Internal state: ', TO_STRING(THIS^.stSeqCtrlGeneral.iInternalSeqStateCase));

E_SEQ_GENERAL.DONE:;

E_SEQ_GENERAL.ERROR:;

E_SEQ_GENERAL.TIME_OUT:; 
IF TRUE
AND THIS^.stSeqCtrlGeneral.bTimeOutActiveQuit 
THEN
  THIS^.stSeqCtrlGeneral.strExtraInfo := 'Bitte quittieren und erneut testen';
  IF TRUE
  //AND itfOpMode.P_QUIT
  THEN
    THIS^.stSeqCtrlGeneral.eActiveSeqState := E_SEQ_GENERAL.EXECUTE;
	END_IF
  
END_IF

ELSE
  THIS^.stSeqCtrlGeneral.eActiveSeqState := E_SEQ_GENERAL.ERROR;
END_CASE
END_METHOD

METHOD PRIVATE _m_SequenceManager
VAR_INPUT
END_VAR
IF FALSE
//AND THIS^.eActiveSeqState=DONE 
AND eLastSeq<>eSeq
THEN
	IF THIS^.stSeqCtrlGeneral.eActiveSeqState<>E_SEQ_GENERAL.EXECUTE THEN
		THIS^.stSeqCtrlGeneral.eActiveSeqState:=E_SEQ_GENERAL.READY;
	END_IF
END_IF

eSeq := eNextSeq;

//DelayTimer und TimeOut Timer verwalten
stSeqCtrlGeneral.bActiveStep:=	TRUE
				AND eLastSeq					=	eSeq
				AND stSeqCtrlGeneral.eLastActiveSeqState			=	stSeqCtrlGeneral.eActiveSeqState
				AND	stSeqCtrlGeneral.iLastInternalSeqStateCase	=	stSeqCtrlGeneral.iInternalSeqStateCase
				;
			
IF NOT stSeqCtrlGeneral.bActiveStep THEN
	stSeqCtrlGeneral.bDelayActive:=FALSE;
	stSeqCtrlGeneral.bTimeOutActiveQuit:=FALSE;
	stSeqCtrlGeneral.bTimeOutActiveNoQuit:=FALSE;
  THIS^.stSeqCtrlGeneral.strExtraInfo:='';
END_IF

_m_SaveLastStep();
stSeqCtrlGeneral.tonDelay	(IN:=stSeqCtrlGeneral.bActiveStep AND stSeqCtrlGeneral.bDelayActive, 		PT:=stSeqCtrlGeneral.tDelay);
stSeqCtrlGeneral.tonTimeOut	(IN:=stSeqCtrlGeneral.bActiveStep AND (stSeqCtrlGeneral.bTimeOutActiveNoQuit OR stSeqCtrlGeneral.bTimeOutActiveQuit), 	PT:=stSeqCtrlGeneral.tTimeOut);
stSeqCtrlGeneral.tonStepTime	(IN:= stSeqCtrlGeneral.bActiveStep, PT:= T#24H);

IF stSeqCtrlGeneral.tonTimeOut.Q  THEN
	stSeqCtrlGeneral.eActiveSeqState:=E_SEQ_GENERAL.TIME_OUT;
END_IF

IF stSeqCtrlGeneral.iError<>0 THEN
	eSeq:=E_SEQ_VALVE.ERROR_SEQ;
END_IF



eLastSeq					:=	eSeq;
stSeqCtrlGeneral.eLastActiveSeqState			:=	stSeqCtrlGeneral.eActiveSeqState;
stSeqCtrlGeneral.iLastInternalSeqStateCase	:=	stSeqCtrlGeneral.iInternalSeqStateCase;

// Reset set ready state
IF THIS^.stSeqCtrlGeneral.bExitSetReadyState THEN
  THIS^.stSeqCtrlGeneral.bExitSetReadyState := FALSE;
END_IF
END_METHOD

METHOD PRIVATE _m_TimeOut : BOOL
VAR_INPUT
	bTimeoutActiveToQuit:	BOOL;
	bTimeOutActiveNoQuit:	BOOL;
	tTimeOut:				TIME;	
END_VAR
THIS^.stSeqCtrlGeneral.bTimeOutActiveQuit:=	bTimeoutActiveToQuit;
THIS^.stSeqCtrlGeneral.bTimeOutActiveNoQuit:=	bTimeOutActiveNoQuit;
THIS^.stSeqCtrlGeneral.tTimeOut:=			tTimeOut;
_m_TimeOut:=FALSE;
IF THIS^.stSeqCtrlGeneral.tonTimeOut.Q THEN
	_m_TimeOut:=TRUE;
END_IF
END_METHOD

METHOD FB_init : BOOL
VAR_INPUT
	bInitRetains : BOOL; // if TRUE, the retain variables are initialized (warm start / cold start)
	bInCopyCode : BOOL;  // if TRUE, the instance afterwards gets moved into the copy code (online change)
  
  itfOpMode:											                        I_OP_MODE; 
  itfEventLogger:                                         I_EVENT_LOGGER;
END_VAR
THIS^.itfOpMode := itfOpMode;
THIS^.itfEventLogger := itfEventLogger;
END_METHOD

METHOD M_Reset : BOOL
VAR_INPUT
END_VAR
M_Reset := THIS^.stSeqCtrlGeneral.eActiveSeqState = E_SEQ_GENERAL.DONE;

// Assign input

// General
IF THIS^.stSeqCtrlGeneral.eActiveSeqState = E_SEQ_GENERAL.READY THEN
  THIS^.eNextSeq := E_SEQ_VALVE.INIT;
  THIS^.stSeqCtrlGeneral.eActiveSeqState := E_SEQ_GENERAL.EXECUTE;
END_IF
END_METHOD

(*=== Method: M_Run  ============================================

 @brief: Here is the global code (Timer, Event, Flange,...)*)
METHOD M_Run
END_METHOD

METHOD M_SetReady : BOOL
VAR_INPUT
END_VAR
M_SetReady := TRUE
              AND THIS^.stSeqCtrlGeneral.eActiveSeqState = E_SEQ_GENERAL.READY
              AND THIS^.eSeq = E_SEQ_VALVE.BASE;

THIS^.stSeqCtrlGeneral.eActiveSeqState := E_SEQ_GENERAL.READY;
THIS^.eNextSeq := E_SEQ_VALVE.BASE;
END_METHOD

METHOD M_ValveCtrl : BOOL
VAR_INPUT
  /// -100 to -1 = Move to HP, 1 to 100 = Move to WP, 0 = Off
  rSpeedInPercent:        REAL;
  tDelay:                 TIME;
END_VAR
M_ValveCtrl := THIS^.stSeqCtrlGeneral.eActiveSeqState = E_SEQ_GENERAL.DONE;

// Assign input
IF rSpeedInPercent < -100 THEN
  rSpeedInPercent := -100;
ELSIF rSpeedInPercent > 100 THEN
  rSpeedInPercent := 100;
END_IF
THIS^.rSpeedInPercent := rSpeedInPercent;
THIS^.tDelay := tDelay;

// General
IF THIS^.stSeqCtrlGeneral.eActiveSeqState = E_SEQ_GENERAL.READY THEN
  THIS^.eNextSeq := E_SEQ_VALVE.SET_LIMIT;
  THIS^.stSeqCtrlGeneral.eActiveSeqState := E_SEQ_GENERAL.EXECUTE;
END_IF
END_METHOD

METHOD M_ValveCtrlSmooth : BOOL
VAR_INPUT
  /// -100 to -1 = Move to HP, 1 to 100 = Move to WP, 0 = Off
  rSpeedInPercent:        REAL;
  tDelay:                 TIME;
END_VAR
M_ValveCtrlSmooth := THIS^.stSeqCtrlGeneral.eActiveSeqState = E_SEQ_GENERAL.DONE;

// Assign input
IF rSpeedInPercent < -100 THEN
  rSpeedInPercent := -100;
ELSIF rSpeedInPercent > 100 THEN
  rSpeedInPercent := 100;
END_IF
THIS^.rSpeedInPercent := rSpeedInPercent;
THIS^.tDelay := tDelay;

// General
IF THIS^.stSeqCtrlGeneral.eActiveSeqState = E_SEQ_GENERAL.READY THEN
  THIS^.eNextSeq := E_SEQ_VALVE.SET_LIMIT_SMOOTH;
  THIS^.stSeqCtrlGeneral.eActiveSeqState := E_SEQ_GENERAL.EXECUTE;
END_IF
END_METHOD

{warning 'Eigenschaftenimplementierung hinzufügen'}
PROPERTY P_CurrentVal : INT
GET
P_CurrentVal := THIS^.iOutputVal;
END_GET
END_PROPERTY

(*=== Property: P_Event  ============================================

 @param [set]: 	Set the Structure "ST_EVENT" from another Object
 @param [get]: 	Return the Structure "ST_EVENT", it contains the actual 
					event of the Object *)
PROPERTY P_Event : GenLib.ST_EVENT
GET
END_GET
SET
END_SET
END_PROPERTY

{warning 'Eigenschaftenimplementierung hinzufügen'}
(*=== Property: P_FullObjectPath  ============================================

 @param [set]: 	Set the Object Path (Clear String of Object)
 @param [get]: 	Return the Objectpath *)
PROPERTY P_FullObjectPath : STRING
GET
END_GET
SET
END_SET
END_PROPERTY

{warning 'Eigenschaftenimplementierung hinzufügen'}
(*=== Property: P_Global_Ack  ============================================

 @param [set]: 	Set the Bit for Ack from another Object
 @param [get]: 	Return the state of Ack Bit*)
PROPERTY P_Global_Ack : BOOL
GET
END_GET
SET
END_SET
END_PROPERTY

{warning 'Eigenschaftenimplementierung hinzufügen'}
(*=== Property: P_GlobalID  ============================================

 @param [set]: 	-
 @param [get]: 	Return the string of instance path*)
PROPERTY P_GlobalID : STRING
GET
END_GET
END_PROPERTY

{warning 'Eigenschaftenimplementierung hinzufügen'}
PROPERTY P_ReadyState : BOOL
GET
P_ReadyState := THIS^.stSeqCtrlGeneral.eActiveSeqState = E_SEQ_GENERAL.READY;
END_GET
END_PROPERTY

PROPERTY P_SpeedInPercent : REAL
GET
P_SpeedInPercent := THIS^.rSpeedInPercent;
END_GET
END_PROPERTY

END_FUNCTION_BLOCK

// ---- MODULE/ACTOR_VALVE/HYDRAULIC_ACTOR/POU/FB_CYLINDER_DA_COUNTER.TcPOU
FUNCTION_BLOCK FB_CYLINDER_DA_COUNTER IMPLEMENTS I_CYLINDER_DA_COUNTER
VAR_INPUT
  //lrCurrentPosAbs:                                        LREAL;
  rCurrentPressureInBar:                                  REAL;
  bJogActive:                                             BOOL;
  rPressureRegulationFactor:                              REAL;
  rPressureRegulationTolerance:                           REAL;
END_VAR
VAR //General
	{attribute 'instance-path'} 
  {attribute 'noinit'} 
	strInstancePath:									                      STRING;
	bInit: 												                          BOOL:=TRUE;
	strFullObjectPath: 								                      STRING;
	stEvent:											                          ST_EVENT;
	bAck:												                            BOOL;
	
END_VAR
VAR   // From FB_init	
	itfOpMode:											                        I_OP_MODE; 
  itfEventLogger:                                         I_EVENT_LOGGER;
  itfOpModeVisu:											                    I_OP_MODE_PAUSE_VISU; 
  itfValve_CylCtrl:                                       I_VALVE_X_3;
  itfValve_Bypass:                                        I_VALVE_X_2;
  itfValve_AutomaticEnable:                               I_VALVE_X_2;
  itfValve_SinkBlock:                                     I_VALVE_X_2;
  itfValve_LowPressureCircuitAdd:                         I_VALVE_X_2;
  itfValve_PressureLimit:                                 I_PRV_PROP;
  itfJogBtnPos_Pressed:                                   I_BINARY_SWITCH;
  itfJogBtnNeg_Pressed:                                   I_BINARY_SWITCH;
  lrPistonSurfaceA:                                       LREAL;
  lrPistonSurfaceB:                                       LREAL;
  rEndPosTol:                                             REAL;
  /// Volume flow in l/min or dm³/min
  rPumpVolumeFlow:                                        REAL; // Volumenstrom
  /// Pump efficiency factor (0,5-1)
  rPumpEfficiencyFactor:                                  REAL; // Wirkungsgrad
END_VAR                                      				
VAR	// Step chain control                				
  eSeq, eLastSeq, eNextSeq:					                      E_SEQ_CYLINDER; 
                  				
  //eActiveSeqState, eLastActiveSeqState:                 E_SEQ_GENERAL;
	(*
  iInternalSeqStateCase, iLastInternalSeqStateCase:       INT:=0;       
	tonDelay, tonTimeOut, tonStepTime:						          TON;
	tDelay:													                        TIME := T#100MS;
	tTimeOut:												                        TIME := T#100MS;
	tTimeOutExt:											                      TIME := T#100MS;
	bDelayActive, bTimeOutActiveQuit, bTimeOutActiveNoQuit:	BOOL;//Timer Option
	bActiveStep, bDebugAcitve, bDebugNext:					        BOOL;//Debug Option
	i:														                          INT;
 	iError:													                        INT; //ERROR-CODE                    	                   		
	listLastSteps:											                    ARRAY[0..49] OF ST_LAST_STEPS;	
	strExtraInfo:											                      STRING; 
	eStep_Type:												                      E_STEP_STATE_TYPE; 
	bDebugModeActive:										                    BOOL;   
	bWaitForBreakpoint:										                  BOOL;
	bBreakpointActive:										                  BOOL;
	bDebugResume:											                      BOOL;   
	listBreakpoint:											                    ARRAY[0..10] OF  INT;    
*)
i:														                            INT;
ii:														                            INT;
iii:														                          INT;
stSeqCtrlGeneral:											                    ST_SEQ_CTRL_GEN;     	
END_VAR                                             		
VAR                                                 		
	bMethodeFromExtStarted:									                BOOL;
	bMethodeFromExtActive:									                BOOL;
	bMethodeFromExtDone:									                  BOOL;
	strTemp:												                        STRING;
END_VAR   
VAR
  stHMI:                                                  ST_HMI_CYLINDER;
  rTargetPressureInBarA:                                  REAL;
  rTargetPressureInBarB:                                  REAL;
  rTargetPressureInForceA:                                REAL;
  rTargetPressureInForceB:                                REAL;
  rTargetPressureInPercentA:                              REAL;
  rTargetPressureInPercentB:                              REAL;
  iTargetPressureAsValueA:                                INT;
  iTargetPressureAsValueB:                                INT;
  rStrokeLength:                                          REAL;
  bJogCtrlBusy:                                           BOOL;
  bStartHPTrigger:                                        BOOL;
  bStartWPTrigger:                                        BOOL;
  bStopTrigger:                                           BOOL;
  bStartSetPosTrigger:                                    BOOL;
  bStartCalibrationClicked:                               BOOL;
  bLowPressureCircuitEnabled:                             BOOL;
  rCurrentForceInKN:                                      REAL;
  rCurrentForceInN:                                       REAL;
  rActiveForce:                                           REAL;
  iCorrectedPressureAsValue:                              INT;
  bRegulationTrigger:                                     BOOL;
  bRegulationBusy:                                        BOOL;
  bCorrectionTrigger:                                     BOOL;
  uiRegulationSeq:                                        UINT := 0;
  bRegulation:                                            BOOL;
END_VAR                  	
VAR_TEMP                    	
	iTemp:										                              INT;
END_VAR
VAR PERSISTENT
	listCylCalibration:                                     ARRAY[1..2, 1..100] OF LREAL;
  listCalibrationTable:                                   ARRAY[1..7] OF ST_CYL_CALIBRATION;
END_VAR

// Set FBs and Interfaces ready after switch internal step
IF stSeqCtrlGeneral.iInternalSeqStateCase <> stSeqCtrlGeneral.iLastInternalSeqStateCase AND NOT stSeqCtrlGeneral.bExitSetReadyState THEN
  IF TRUE
  AND itfValve_CylCtrl.M_SetReady()
  AND itfValve_Bypass.M_SetReady()
  AND itfValve_AutomaticEnable.M_SetReady()
  AND itfValve_SinkBlock.M_SetReady()
  AND itfValve_LowPressureCircuitAdd.M_SetReady()
  AND itfValve_PressureLimit.M_SetReady()
  THEN
    stSeqCtrlGeneral.bExitSetReadyState := TRUE;
  ELSE
    RETURN;
  END_IF
END_IF

stSeqCtrlGeneral.strObjectPath := strInstancePath;
stSeqCtrlGeneral.strObject := F_CreateObjectName(strInstancePath);

// Calibration table
FOR iii := 1 TO 7 BY 1 DO
  listCylCalibration[2, iii] := TO_LREAL(listCalibrationTable[iii].uiValue);
  listCylCalibration[1, iii] := TO_LREAL(listCalibrationTable[iii].uiPressure);
END_FOR

rCurrentForceInKN := P_CurrentForceInKN;
rCurrentForceInN := P_CurrentForceInKN * 1000;

// First method call
_m_SequenceManager();
//_m_SaveLastStep();
_m_ManualOperation();
_m_PressureCalibration();
_m_PressureRegulation();
_m_HMI();

CASE eSeq OF 
  E_SEQ_CYLINDER.BASE:;
  
	E_SEQ_CYLINDER.INIT: _m_Seq_INIT();
		IF TRUE
		AND (stSeqCtrlGeneral.eActiveSeqState = E_SEQ_GENERAL.DONE) 
		THEN
			eSeq := E_SEQ_CYLINDER.BASE;
		END_IF
		
	E_SEQ_CYLINDER.SETUP:;
  
	// Process
  E_SEQ_CYLINDER.SET_WORK_PRESSURE: _m_Seq_SET_WORK_PRESSURE();
    IF TRUE
		AND (stSeqCtrlGeneral.eActiveSeqState = E_SEQ_GENERAL.DONE) 
		THEN
			eSeq := E_SEQ_CYLINDER.BASE;
		END_IF
  
  E_SEQ_CYLINDER.STOP: _m_Seq_STOP();
    IF TRUE
		AND (stSeqCtrlGeneral.eActiveSeqState = E_SEQ_GENERAL.DONE) 
		THEN
			eSeq := E_SEQ_CYLINDER.BASE;
		END_IF
  
  E_SEQ_CYLINDER.TO_HP: _m_Seq_TO_HP();
    IF TRUE
		AND (stSeqCtrlGeneral.eActiveSeqState = E_SEQ_GENERAL.DONE) 
		THEN
			eSeq := E_SEQ_CYLINDER.BASE;
		END_IF
  
  E_SEQ_CYLINDER.TO_WP: _m_Seq_TO_WP();
    IF TRUE
		AND (stSeqCtrlGeneral.eActiveSeqState = E_SEQ_GENERAL.DONE) 
		THEN
			eSeq := E_SEQ_CYLINDER.BASE;
		END_IF
    
  E_SEQ_CYLINDER.PRESSURE_CALIBRATION: _m_Seq_PRESSURE_CALIBRATION();
    IF TRUE
		AND (stSeqCtrlGeneral.eActiveSeqState = E_SEQ_GENERAL.DONE) 
		THEN
			eSeq := E_SEQ_CYLINDER.BASE;
		END_IF
    
  E_SEQ_CYLINDER.LOW_PRESSURE_CIRCUIT: _m_Seq_LOW_PRESSURE_CIRCUIT();
    IF TRUE
		AND (stSeqCtrlGeneral.eActiveSeqState = E_SEQ_GENERAL.DONE) 
		THEN
			eSeq := E_SEQ_CYLINDER.BASE;
		END_IF

  // End
	E_SEQ_CYLINDER.END:;
	E_SEQ_CYLINDER.ERROR_SEQ:;	
END_CASE

strTemp:=TO_STRING(eSeq);

METHOD PRIVATE _m_DebugManager
VAR_INPUT
	iStepID: int;
END_VAR
IF TRUE
AND THIS^.stSeqCtrlGeneral.bDebugModeActive 
AND NOT THIS^.stSeqCtrlGeneral.bActiveStep
THEN


THIS^.stSeqCtrlGeneral.bBreakpointActive:=FALSE;

FOR i:=0 TO 10 DO
	
	IF TRUE
	AND iStepID=THIS^.stSeqCtrlGeneral.listBreakpoint[i] 
	AND iStepID<>0
	THEN
		EXIT;
	END_IF
END_FOR
IF (i<=10) THEN
	THIS^.stSeqCtrlGeneral.bBreakpointActive:=TRUE;
END_IF

END_IF
END_METHOD

METHOD PRIVATE _m_Delay : BOOL
VAR_INPUT
	DelayTime:	TIME;
END_VAR
THIS^.stSeqCtrlGeneral.bDelayActive:=TRUE;
THIS^.stSeqCtrlGeneral.tDelay:=DelayTime;
_m_Delay:=FALSE;
IF THIS^.stSeqCtrlGeneral.tonDelay.Q THEN
	_m_Delay:=TRUE;
END_IF
END_METHOD

METHOD PRIVATE _m_GeneralStepSetting : BOOL
VAR_INPUT
	StepType:			    	E_STEP_STATE_TYPE;
	InfoTextID:					STRING(20);
	EnableDebug:	   			BOOL;	
	
END_VAR
IF THIS^.stSeqCtrlGeneral.bActiveStep THEN
	THIS^.stSeqCtrlGeneral.eStep_Type:=StepType;
	THIS^.stSeqCtrlGeneral.strExtraInfo:= GenLib.F_RET_TXTLIST_ENTRY(strPortNr:='851',strID:='',strTxtLstName:=InfoTextID);
END_IF
END_METHOD

METHOD PRIVATE _m_HMI : BOOL
VAR_INPUT
END_VAR
// HMI
//stHMI.bInHP := P_Position <= P_MinPosVal + 1;
//stHMI.bInWP := P_Position >= P_MaxPosVal - 1;
//stHMI.bPressureOk := P_PressureOk;
//stHMI.lrCurrentPos := P_Position;
//stHMI.lrMaxPosVal := P_MaxPosVal;
//stHMI.lrMinPosVal := P_MinPosVal;
//stHMI.lrPosToSet := lrToSetPos;
THIS^.stHMI.sState := TO_STRING(THIS^.eSeq);
//stHMI.uiSpeedInPercent
END_METHOD

METHOD PRIVATE _m_ManualOperation : BOOL
VAR_INPUT
END_VAR
IF TRUE 
AND THIS^.itfOpMode.P_OP_MODE_STATE = OP_MODE.MANUAL 
AND THIS^.itfOpModeVisu.P_HandSelected
AND THIS^.stHMI.bToHPTriggered
AND NOT THIS^.bJogCtrlBusy
THEN
  THIS^.stSeqCtrlGeneral.eActiveSeqState := E_SEQ_GENERAL.READY;
  THIS^.bStartHPTrigger := TRUE;
  THIS^.bJogCtrlBusy := TRUE;
ELSIF TRUE 
AND THIS^.itfOpMode.P_OP_MODE_STATE = OP_MODE.MANUAL 
AND THIS^.itfOpModeVisu.P_HandSelected
AND THIS^.stHMI.bToWPTriggered
AND NOT THIS^.bJogCtrlBusy
THEN
  THIS^.stSeqCtrlGeneral.eActiveSeqState := E_SEQ_GENERAL.READY;
  THIS^.bStartWPTrigger := TRUE;
  THIS^.bJogCtrlBusy := TRUE; 
ELSIF TRUE 
AND THIS^.itfOpMode.P_OP_MODE_STATE = OP_MODE.MANUAL 
AND THIS^.itfOpModeVisu.P_HandSelected
AND THIS^.stHMI.bToSetPosTriggered
AND NOT THIS^.bJogCtrlBusy
THEN
  //M_ToSetPos(lrToSetPos:= 500, rSpeedInPercent:= 100);
  THIS^.bJogCtrlBusy := TRUE;
ELSIF TRUE 
AND THIS^.itfOpMode.P_OP_MODE_STATE = OP_MODE.MANUAL 
AND THIS^.itfOpModeVisu.P_HandSelected
AND NOT THIS^.stHMI.bToHPTriggered
AND NOT THIS^.stHMI.bToWPTriggered
AND NOT THIS^.stHMI.bToSetPosTriggered
AND THIS^.bJogCtrlBusy
THEN
  THIS^.stSeqCtrlGeneral.eActiveSeqState := E_SEQ_GENERAL.READY;
  THIS^.bStopTrigger := TRUE;
  THIS^.bStartHPTrigger := FALSE;
  THIS^.bStartWPTrigger := FALSE;
  THIS^.bJogCtrlBusy := FALSE;
END_IF

// JOG
IF TRUE 
AND THIS^.itfOpMode.P_OP_MODE_STATE = OP_MODE.MANUAL 
AND THIS^.itfOpModeVisu.P_JogSelected
THEN
  IF TRUE
  AND THIS^.bJogActive
  AND THIS^.itfJogBtnPos_Pressed.P_Active
  AND NOT THIS^.bJogCtrlBusy
  THEN
    THIS^.stSeqCtrlGeneral.eActiveSeqState := E_SEQ_GENERAL.READY;
    THIS^.bStartWPTrigger := TRUE;
    THIS^.bJogCtrlBusy := TRUE; 
  ELSIF TRUE
  AND THIS^.bJogActive
  AND THIS^.itfJogBtnNeg_Pressed.P_Active
  AND NOT THIS^.bJogCtrlBusy
  THEN
    THIS^.stSeqCtrlGeneral.eActiveSeqState := E_SEQ_GENERAL.READY;
    THIS^.bStartHPTrigger := TRUE;
    THIS^.bJogCtrlBusy := TRUE; 
  ELSIF TRUE
  AND NOT THIS^.itfJogBtnPos_Pressed.P_Active
  AND NOT THIS^.itfJogBtnNeg_Pressed.P_Active
  AND THIS^.bJogCtrlBusy
  THEN
    THIS^.stSeqCtrlGeneral.eActiveSeqState := E_SEQ_GENERAL.READY;
    THIS^.bStopTrigger := TRUE;
    THIS^.bStartHPTrigger := FALSE;
    THIS^.bStartWPTrigger := FALSE;
    THIS^.bJogCtrlBusy := FALSE;
	END_IF
END_IF



IF THIS^.bStartWPTrigger THEN
  IF M_ToWP(ePressureType:= E_PRESSURE_TYPE.BAR, 
            rWorkPressure:= 20, 
            bPressureRegulation:= FALSE,
            eSpeedType:= E_SPEED_TYPE.PERCENT, 
            rSpeed:= 100) THEN
    THIS^.bStartWPTrigger := FALSE;
	END_IF
END_IF
IF THIS^.bStartHPTrigger THEN
  IF M_ToHP(ePressureType:= E_PRESSURE_TYPE.BAR, 
            rWorkPressure:= 20, 
            bPressureRegulation:= FALSE,
            eSpeedType:= E_SPEED_TYPE.PERCENT, 
            rSpeed:= 100) THEN
    THIS^.bStartHPTrigger := FALSE;
	END_IF
END_IF
IF THIS^.bStopTrigger THEN
  IF M_Stop() THEN
    THIS^.bStopTrigger := FALSE;
	END_IF
END_IF
END_METHOD

METHOD PRIVATE _m_PressureCalibration : BOOL
VAR_INPUT
END_VAR
// Calibration clicked
IF TRUE
AND THIS^.itfOpMode.P_OP_MODE_STATE = OP_MODE.MANUAL 
AND THIS^.bStartCalibrationClicked 
THEN
  IF M_PressureCalibration() THEN
    THIS^.stSeqCtrlGeneral.eActiveSeqState := E_SEQ_GENERAL.READY;
    THIS^.bStartCalibrationClicked := FALSE;
	END_IF
END_IF
END_METHOD

(******************Description****************)
// This function allows variable pressure control
(*********************************************)
METHOD PRIVATE _m_PressureRegulation : BOOL
VAR_INPUT
END_VAR
IF TRUE
AND THIS^.rCurrentForceInN < THIS^.rActiveForce 
AND THIS^.iCorrectedPressureAsValue < 32768
AND THIS^.bRegulationTrigger
AND NOT THIS^.bRegulationBusy
THEN
  IF ABS(THIS^.rCurrentForceInN - THIS^.rActiveForce) > THIS^.rPressureRegulationTolerance THEN
    //THIS^.iCorrectedPressureAsValue := THIS^.iCorrectedPressureAsValue + 100;
    THIS^.iCorrectedPressureAsValue := TO_INT(THIS^.iCorrectedPressureAsValue + ABS((THIS^.rCurrentForceInN - THIS^.rActiveForce) * THIS^.rPressureRegulationFactor));
    THIS^.bCorrectionTrigger := TRUE;
  END_IF
ELSIF TRUE
AND THIS^.rCurrentForceInN > THIS^.rActiveForce 
AND THIS^.iCorrectedPressureAsValue > 0
AND THIS^.bRegulationTrigger
AND NOT THIS^.bRegulationBusy
THEN
  IF ABS(THIS^.rCurrentForceInN - THIS^.rActiveForce) > THIS^.rPressureRegulationTolerance THEN
    //THIS^.iCorrectedPressureAsValue := THIS^.iCorrectedPressureAsValue - 100;
    THIS^.iCorrectedPressureAsValue := TO_INT(THIS^.iCorrectedPressureAsValue - ABS((THIS^.rCurrentForceInN - THIS^.rActiveForce) * THIS^.rPressureRegulationFactor));
    THIS^.bCorrectionTrigger := TRUE;
  END_IF
END_IF

// Set Valve value correction
IF THIS^.bCorrectionTrigger THEN
  THIS^.bRegulationBusy:= TRUE;
  CASE THIS^.uiRegulationSeq OF
    0:;
      IF THIS^.itfValve_PressureLimit.M_SetReady() THEN
        THIS^.uiRegulationSeq := 1;
	    END_IF
    1:;
      IF THIS^.itfValve_PressureLimit.M_SetLimit(ePressureType:= E_PRESSURE_TYPE.VALUE, rLimit:= iCorrectedPressureAsValue) THEN
        THIS^.bCorrectionTrigger := FALSE;
        THIS^.bRegulationBusy := FALSE;
        THIS^.uiRegulationSeq := 0;
	    END_IF
	END_CASE
END_IF
END_METHOD

METHOD PRIVATE _m_SaveLastStep : BOOL
VAR_INPUT
END_VAR
VAR
	i: dint;
END_VAR
IF NOT THIS^.stSeqCtrlGeneral.bActiveStep THEN
	
	FOR i:=49 TO 1 BY -1 DO
			stSeqCtrlGeneral.listLastSteps[i].strStepName:=stSeqCtrlGeneral.listLastSteps[i-1].strStepName;
			stSeqCtrlGeneral.listLastSteps[i].tStepTime:=stSeqCtrlGeneral.listLastSteps[i-1].tStepTime;
			stSeqCtrlGeneral.listLastSteps[i].tDelayTime:=stSeqCtrlGeneral.listLastSteps[i-1].tDelayTime;
	END_FOR
	stSeqCtrlGeneral.listLastSteps[0].strStepName:=TO_STRING(THIS^.eSeq);
	stSeqCtrlGeneral.listLastSteps[1].tStepTime:=THIS^.stSeqCtrlGeneral.tonStepTime.ET;
	stSeqCtrlGeneral.listLastSteps[1].tStepTime:=THIS^.stSeqCtrlGeneral.tonDelay.ET;
ELSE
	stSeqCtrlGeneral.listLastSteps[0].tStepTime:=THIS^.stSeqCtrlGeneral.tonStepTime.ET;
	stSeqCtrlGeneral.listLastSteps[0].tDelayTime:=THIS^.stSeqCtrlGeneral.tonDelay.ET;	
END_IF
END_METHOD

METHOD PRIVATE _m_Seq_INIT : E_SEQ_PROCESS
VAR_INPUT
END_VAR
VAR
	ActiveSeq: STRING;
END_VAR
VAR
	
END_VAR
//THIS^._m_GeneralStepSetting(StepType:=E_STEP_STATE_TYPE.INIT,
ActiveSeq := TO_STRING(THIS^.eSeq);

CASE THIS^.stSeqCtrlGeneral.eActiveSeqState OF
E_SEQ_GENERAL.READY:;

	
E_SEQ_GENERAL.EXECUTE:;
	IF TRUE
	THEN
		THIS^.stSeqCtrlGeneral.eActiveSeqState := E_SEQ_GENERAL.RESET;
	END_IF
E_SEQ_GENERAL.RESET:;
	stSeqCtrlGeneral.iInternalSeqStateCase := 0;
	IF TRUE
	THEN
		THIS^.stSeqCtrlGeneral.eActiveSeqState := E_SEQ_GENERAL.BUSY;
	END_IF
E_SEQ_GENERAL.BUSY:;
	CASE THIS^.stSeqCtrlGeneral.iInternalSeqStateCase OF
		0:	// Reset valves
      IF TRUE
      AND THIS^.itfValve_AutomaticEnable.M_ToHP(tDelay:= T#10MS)
      AND THIS^.itfValve_Bypass.M_ToHP(tDelay:= T#10MS)
      AND THIS^.itfValve_CylCtrl.M_ToHP(tDelay:= T#10MS)
      AND THIS^.itfValve_LowPressureCircuitAdd.M_ToHP(tDelay:= T#10MS)
      AND THIS^.itfValve_SinkBlock.M_ToHP(tDelay:= T#10MS)
			THEN 
				THIS^.stSeqCtrlGeneral.iInternalSeqStateCase := 1000;
			END_IF
      
    1000: // Exit step
      IF TRUE
			THEN 
				THIS^.stSeqCtrlGeneral.iInternalSeqStateCase := 9999;
			END_IF
      
	ELSE
		THIS^.stSeqCtrlGeneral.eActiveSeqState := E_SEQ_GENERAL.DONE;  
	END_CASE
	THIS^.stSeqCtrlGeneral.strExtraInfo := CONCAT('Internal state: ', TO_STRING(THIS^.stSeqCtrlGeneral.iInternalSeqStateCase));
E_SEQ_GENERAL.DONE:;
E_SEQ_GENERAL.ERROR:;
E_SEQ_GENERAL.TIME_OUT:; 

IF TRUE
AND THIS^.stSeqCtrlGeneral.bTimeOutActiveQuit 
THEN
  THIS^.stSeqCtrlGeneral.strExtraInfo := 'Bitte quittieren und erneut testen';
  IF TRUE
  //AND itfOpMode.P_QUIT
  THEN
    THIS^.stSeqCtrlGeneral.eActiveSeqState := E_SEQ_GENERAL.EXECUTE;
	END_IF
  
END_IF

ELSE
  THIS^.stSeqCtrlGeneral.eActiveSeqState := E_SEQ_GENERAL.ERROR;
END_CASE
END_METHOD

METHOD PRIVATE _m_Seq_LOW_PRESSURE_CIRCUIT : E_SEQ_PROCESS
VAR_INPUT
END_VAR
VAR
	ActiveSeq: STRING;
END_VAR
VAR
	
END_VAR
//THIS^._m_GeneralStepSetting(StepType:=E_STEP_STATE_TYPE.INIT,
ActiveSeq := TO_STRING(THIS^.eSeq);

CASE THIS^.stSeqCtrlGeneral.eActiveSeqState OF
E_SEQ_GENERAL.READY:;

	
E_SEQ_GENERAL.EXECUTE:;
	IF TRUE
  //AND _m_Delay(DelayTime:= T#10MS)
	THEN
		THIS^.stSeqCtrlGeneral.eActiveSeqState := E_SEQ_GENERAL.RESET;
	END_IF
  
E_SEQ_GENERAL.RESET:;
	stSeqCtrlGeneral.iInternalSeqStateCase := 0;
	IF TRUE
	THEN
		THIS^.stSeqCtrlGeneral.eActiveSeqState := E_SEQ_GENERAL.BUSY;
	END_IF
  
E_SEQ_GENERAL.BUSY:;
	CASE THIS^.stSeqCtrlGeneral.iInternalSeqStateCase OF
		0: // Switch off valves
      IF TRUE
			THEN 
        IF THIS^.bLowPressureCircuitEnabled THEN
          THIS^.stSeqCtrlGeneral.iInternalSeqStateCase := 10;
        ELSE
          THIS^.stSeqCtrlGeneral.iInternalSeqStateCase := 20;
				END_IF
			END_IF
      
    10: // Add low pressure circuit
      IF TRUE
      AND THIS^.itfValve_LowPressureCircuitAdd.M_ToWP1(tDelay:= T#0MS)
			THEN 
        THIS^.stSeqCtrlGeneral.iInternalSeqStateCase := 1000;
			END_IF
      
    20: // Disable low pressure circuit
      IF TRUE
      AND THIS^.itfValve_LowPressureCircuitAdd.M_ToHP(tDelay:= T#0MS)
			THEN 
        THIS^.stSeqCtrlGeneral.iInternalSeqStateCase := 1000;
			END_IF
      
    1000: // Exit step
      IF TRUE
			THEN 
				THIS^.stSeqCtrlGeneral.iInternalSeqStateCase := 9999;
			END_IF
      
	ELSE
		THIS^.stSeqCtrlGeneral.eActiveSeqState := E_SEQ_GENERAL.DONE;  
	END_CASE
	THIS^.stSeqCtrlGeneral.strExtraInfo := CONCAT('Internal state: ', TO_STRING(THIS^.stSeqCtrlGeneral.iInternalSeqStateCase));

E_SEQ_GENERAL.DONE:;

E_SEQ_GENERAL.ERROR:;

E_SEQ_GENERAL.TIME_OUT:; 
IF TRUE
AND THIS^.stSeqCtrlGeneral.bTimeOutActiveQuit 
THEN
  THIS^.stSeqCtrlGeneral.strExtraInfo := 'Bitte quittieren und erneut testen';
  IF TRUE
  //AND itfOpMode.P_QUIT
  THEN
    THIS^.stSeqCtrlGeneral.eActiveSeqState := E_SEQ_GENERAL.EXECUTE;
	END_IF
  
END_IF

